// TwinCAT 3 PLC project plc_kfe_gatt
// Title: KFE GATT
// Company: LCLS - ECS
// ProjectVersion: 0.3.1
// ProgramVersion: 3.1.4023.0
// CompilerDefines: K
// libraries:
//   LCLS General, * (SLAC)
//   LCLS Vacuum, * (SLAC - LCLS)
//   lcls-twincat-motion, * (SLAC)
//   PMPS, * (SLAC - LCLS)
//   Tc2_ControllerToolbox, * (Beckhoff Automation GmbH)
//   Tc2_EtherCAT, * (Beckhoff Automation GmbH)
//   Tc2_MC2, * (Beckhoff Automation GmbH)
//   Tc2_Standard, * (Beckhoff Automation GmbH)
//   Tc2_System, * (Beckhoff Automation GmbH)
//   Tc2_Utilities, * (Beckhoff Automation GmbH)
//   Tc3_JsonXml, * (Beckhoff Automation GmbH)
//   Tc3_Module, * (Beckhoff Automation GmbH)
//   TcUnit, * (www.tcunit.org)
// project tree:
//   DUTs/ E_State.TcDUT, E_GasType.TcDUT, E_HomeState.TcDUT, E_MAA_States.TcDUT, E_MAA_States_X.TcDUT, E_MoveState.TcDUT, ST_DRL.TcDUT, ST_VGP.TcDUT
//   Version/ Global_Version.TcGVL
//   GVLs/ GVL_Devices.TcGVL, GVL_GATT.TcGVL, GVL_PMPS.TcGVL, GVL_MOT.TcGVL, GVL_Variables.TcGVL, Main.TcGVL
//   / PlcTask.TcTTO
//   POUs/ DIAGNOSTICS.TcPOU, FB_MAA.TcPOU, FB_MAA_States.TcPOU, FB_MAA_States_X.TcPOU, FB_VGP.TcPOU, PRG_1_PlcTask.TcPOU, PRG_GasSelection.TcPOU, PRG_GATT.TcPOU, PRG_ILK.TcPOU, PRG_INJ.TcPOU, PRG_Motion.TcPOU, PRG_Motors_Test.TcPOU, PRG_PMPS.TcPOU, PRG_Transmission.TcPOU, PRG_VGP.TcPOU
//   POUs/Test/ FB_ILK_TEST.TcPOU, FB_VCN_Lin.TcPOU
//   POUs/Transmission/ F_COEF_AR.TcPOU
// real-time tasks:
//   TASK PlcTask: cycle T#10ms, priority 20, ADS port 350
// motion (NC):
//   TASK NC-Task 1 SAF: cycle T#2ms, priority 4, ADS port 501
//   TASK NC-Task 1 SVB: cycle T#10ms, priority 8, ADS port 511
//   AXIS MA_1_X (id 1)
//     Velo: Maximum=1
//     OtherSettings: AllowMotionCmdToSlave=true
//     encoder EncType=7
//       EncPara: ScaleFactorNumerator=0.000117010498, Offset=1.88, Inverse=true, MaxCount=#x0000ffff, ReferenceSystem=1
//         SoftEndMinControl: Enable=true, Range=-2
//         SoftEndMaxControl: Enable=true, Range=2
//         Inc: RefSoftSyncMask=#x0000ffff
//     drive DrvType=24
//       Analog: VeloReferenz=7.93496, TorqueScale=10, ScaleFactorActTorque=0.1
//       TimeComp: TaskDelayCycles=1
//     controller CtrType=1
//       CtrPara: PriorControlFactor=1
//         PosDiffControl: Range=0.2
//         Observer: BandWidth=20
//   AXIS MA_1_Y (id 2)
//     Dynamic: AccelerationMaximum=30, DecelerationMaximum=30
//     Velo: Maximum=10
//     TargetPosControl: Range=0.5
//     OtherSettings: AllowMotionCmdToSlave=true
//     encoder EncType=7
//       EncPara: ScaleFactorNumerator=0.001490478515625, Offset=-48.83, MaxCount=#x0000ffff, ReferenceSystem=1
//         SoftEndMinControl: Enable=true, Range=-48.8
//         SoftEndMaxControl: Enable=true
//         Inc: RefSoftSyncMask=#x0000ffff
//     drive DrvType=24
//       Analog: VeloReferenz=40, TorqueScale=10, ScaleFactorActTorque=0.1
//       TimeComp: TaskDelayCycles=1
//     controller CtrType=1
//       CtrPara: PriorControlFactor=1
//         PosDiffControl: Range=0.5
//         Observer: BandWidth=20
//   AXIS MA_2_X (id 3)
//     Velo: Maximum=1
//     OtherSettings: AllowMotionCmdToSlave=true
//     encoder EncType=7
//       EncPara: ScaleFactorNumerator=7.6080322266e-05, Offset=-0.496, MaxCount=#x0000ffff, ReferenceSystem=1
//         SoftEndMinControl: Enable=true, Range=-1.59
//         SoftEndMaxControl: Enable=true, Range=1.59
//         Inc: RefSoftSyncMask=#x0000ffff
//     drive DrvType=24
//       Analog: VeloReferenz=7.93496, TorqueScale=10, ScaleFactorActTorque=0.1
//       TimeComp: TaskDelayCycles=1
//     controller CtrType=1
//       CtrPara: PriorControlFactor=1
//         PosDiffControl: Range=0.1
//         Observer: BandWidth=20
//   AXIS MA_2_Y (id 4)
//     Dynamic: AccelerationMaximum=30, DecelerationMaximum=30
//     Velo: Maximum=10
//     TargetPosControl: Range=0.5
//     OtherSettings: AllowMotionCmdToSlave=true
//     encoder EncType=7
//       EncPara: ScaleFactorNumerator=0.001524353027344, Offset=-49.38, MaxCount=#x0000ffff, ReferenceSystem=1
//         SoftEndMinControl: Enable=true, Range=-48.99
//         SoftEndMaxControl: Enable=true
//         Inc: RefSoftSyncMask=#x0000ffff
//     drive DrvType=24
//       Analog: VeloReferenz=50, TorqueScale=10, ScaleFactorActTorque=0.1
//       TimeComp: TaskDelayCycles=1
//     controller CtrType=1
//       CtrPara: PriorControlFactor=1
//         PosDiffControl: Range=0.5
//         Observer: BandWidth=20
//   AXIS MA_3_X (id 5)
//     Velo: Maximum=1
//     OtherSettings: AllowMotionCmdToSlave=true
//     encoder EncType=7
//       EncPara: ScaleFactorNumerator=0.0001220703125, Offset=-2.029, MaxCount=#x0000ffff, ReferenceSystem=1
//         SoftEndMinControl: Enable=true, Range=-1.6
//         SoftEndMaxControl: Enable=true, Range=1.6
//         Inc: RefSoftSyncMask=#x0000ffff
//     drive DrvType=24
//       Analog: VeloReferenz=7.93496, TorqueScale=10, ScaleFactorActTorque=0.1
//       TimeComp: TaskDelayCycles=1
//     controller CtrType=1
//       CtrPara: PriorControlFactor=1
//         PosDiffControl: Range=0.1
//         Observer: BandWidth=20
//   AXIS MA_3_Y (id 6)
//     Dynamic: AccelerationMaximum=30, DecelerationMaximum=30
//     Velo: Maximum=10
//     TargetPosControl: Range=0.5
//     OtherSettings: AllowMotionCmdToSlave=true
//     encoder EncType=7
//       EncPara: ScaleFactorNumerator=0.001514892578125, Offset=-49.49, MaxCount=#x0000ffff, ReferenceSystem=1
//         SoftEndMinControl: Enable=true, Range=-49.27
//         SoftEndMaxControl: Enable=true
//         Inc: RefSoftSyncMask=#x0000ffff
//     drive DrvType=24
//       Analog: VeloReferenz=50, TorqueScale=10, ScaleFactorActTorque=0.1
//       TimeComp: TaskDelayCycles=1
//     controller CtrType=1
//       CtrPara: PriorControlFactor=1
//         PosDiffControl: Range=0.2
//         Observer: BandWidth=20
//   AXIS MA_4_X (id 7)
//     Velo: Maximum=1
//     OtherSettings: AllowMotionCmdToSlave=true
//     encoder EncType=7
//       EncPara: ScaleFactorNumerator=0.0001022338867, Offset=-1.581, MaxCount=#x0000ffff, ReferenceSystem=1
//         SoftEndMinControl: Enable=true, Range=-1.58
//         SoftEndMaxControl: Enable=true, Range=1.76
//         Inc: RefSoftSyncMask=#x0000ffff
//     drive DrvType=24
//       Analog: VeloReferenz=7.93496, TorqueScale=10, ScaleFactorActTorque=0.1
//       TimeComp: TaskDelayCycles=1
//     controller CtrType=1
//       CtrPara: PriorControlFactor=1
//         PosDiffControl: Range=0.2
//         Observer: BandWidth=20
//   AXIS MA_4_Y (id 8)
//     Dynamic: AccelerationMaximum=30, DecelerationMaximum=30
//     Velo: Maximum=10
//     TargetPosControl: Range=0.5
//     OtherSettings: AllowMotionCmdToSlave=true
//     encoder EncType=7
//       EncPara: ScaleFactorNumerator=0.001497802734375, Offset=-49.07, MaxCount=#x0000ffff, ReferenceSystem=1
//         SoftEndMinControl: Enable=true, Range=-49.08
//         SoftEndMaxControl: Enable=true, Range=0.009
//         Inc: RefSoftSyncMask=#x0000ffff
//     drive DrvType=24
//       Analog: VeloReferenz=50, TorqueScale=10, ScaleFactorActTorque=0.1
//       TimeComp: TaskDelayCycles=1
//     controller CtrType=1
//       CtrPara: PriorControlFactor=1
//         PosDiffControl: Range=0.2
//         Observer: BandWidth=20
//   AXIS VGP_80 (id 9)
//     Velo: Maximum=1800
//     OtherSettings: AllowMotionCmdToSlave=true
//     encoder EncType=4
//       EncPara: ScaleFactorNumerator=0.0390625, Inverse=true, MaxCount=#x0000ffff
//         SoftEndMinControl: Enable=true, Range=-15
//         SoftEndMaxControl: Enable=true, Range=1680
//         Inc: RefSoftSyncMask=#x0000ffff
//     drive DrvType=24
//       Analog: VeloReferenz=1000, TorqueScale=10, ScaleFactorActTorque=0.1
//       TimeComp: TaskDelayCycles=1
//     controller CtrType=1
//       CtrPara: PriorControlFactor=1
//         PosDiffControl: Range=10
//         Observer: BandWidth=20
// I/O:
//   DEVICE =+-CX2020/EtherCAT1, AmsNetId 172.21.92.57.2.1
//     =+-EK1200_00_00 [EK1200-5000 EtherCAT Power supply (2A E-Bus)]
//       =+-ES3064_00_01 [EL3064 4Ch. Ana. Input 0-10V]
//       =+-EL6070_00_02 [EL6070 1Ch. Licensing-Terminal]
//       =+-ES1008_00_03 [EL1008 8Ch. Dig. Input 24V, 3ms]
//       =+-ES2008_00_05 [EL2008 8Ch. Dig. Output 24V, 0.5A]
//       =+-EL2794_00_06 [EL2794 4Ch. Dig. Output 24V AC/DC, 2A, short-circuit-proof]
//       =+-ES2202_00_07 [EL2202 2Ch. Dig. Output 24V, 0.5A]
//       PMPS_PRE [EL6695 EtherCAT Bridge terminal (Primary)]
//       =+-EK1110_00_09 [EK1110 EtherCAT extension]
//     =+-EK1100_01_00 [EK1100 EtherCAT Coupler (2A E-Bus)]
//       =+-ES3064_01_01 [EL3064 4Ch. Ana. Input 0-10V]
//       =+-ES3064_01_02 [EL3064 4Ch. Ana. Input 0-10V]
//       =+-EL2798_01_03 [EL2798 8Ch. Dig. Output 24V AC/DC, 2A, potential-free]
//       =+-ES3064_01_04 [EL3064 4Ch. Ana. Input 0-10V]
//       =+-ES3064_01_05 [EL3064 4Ch. Ana. Input 0-10V]
//       =+-ES3064_01_06 [EL3064 4Ch. Ana. Input 0-10V]
//       =+-ES3064_01_07 [EL3064 4Ch. Ana. Input 0-10V]
//       =+-EL2798_01_08 [EL2798 8Ch. Dig. Output 24V AC/DC, 2A, potential-free]
//       =+-ES3064_01_09 [EL3064 4Ch. Ana. Input 0-10V]
//       =+-ES3064_01_10 [EL3064 4Ch. Ana. Input 0-10V]
//       =+-EL9410_01_11 [EL9410 E-Bus Power Supplier  (Diagnostics)]
//       =+-ES3064_01_12 [EL3064 4Ch. Ana. Input 0-10V]
//       =+-ES3064_01_13 [EL3064 4Ch. Ana. Input 0-10V]
//       =+-EL2798_01_14 [EL2798 8Ch. Dig. Output 24V AC/DC, 2A, potential-free]
//       =+-ES3064_01_15 [EL3064 4Ch. Ana. Input 0-10V]
//       =+-ES3064_01_16 [EL3064 4Ch. Ana. Input 0-10V]
//       =+-ES3064_01_17 [EL3064 4Ch. Ana. Input 0-10V]
//       =+-ES3064_01_18 [EL3064 4Ch. Ana. Input 0-10V]
//       =+-EL2798_01_19 [EL2798 8Ch. Dig. Output 24V AC/DC, 2A, potential-free]
//       =+-ES3064_01_20 [EL3064 4Ch. Ana. Input 0-10V]
//       =+-ES3064_01_21 [EL3064 4Ch. Ana. Input 0-10V]
//       =+-EK1110_01_22 [EK1110 EtherCAT extension]
//     =+-EK1100_02_00 [EK1100 EtherCAT Coupler (2A E-Bus)]
//       =+-ES2004_02_01 [EL2004 4Ch. Dig. Output 24V, 0.5A]
//       =+-ES1004_02_02 [EL1004 4Ch. Dig. Input 24V, 3ms]
//       =+-ES2004_02_03 [EL2004 4Ch. Dig. Output 24V, 0.5A]
//       =+-ES1004_02_04 [EL1004 4Ch. Dig. Input 24V, 3ms]
//       =+-ES7041_02_05 [EL7041 1Ch. Stepper motor output stage (50V, 5A)]
//       =+-ES7041_02_06 [EL7041 1Ch. Stepper motor output stage (50V, 5A)]
//       =+-ES2004_02_07 [EL2004 4Ch. Dig. Output 24V, 0.5A]
//       =+-ES1004_02_08 [EL1004 4Ch. Dig. Input 24V, 3ms]
//       =+-ES7041_02_09 [EL7041 1Ch. Stepper motor output stage (50V, 5A)]
//       =+-ES7041_02_10 [EL7041 1Ch. Stepper motor output stage (50V, 5A)]
//       =+-ES3064_02_11 [EL3064 4Ch. Ana. Input 0-10V]
//       =+-ES9070_02_12 [EL9070 Shield terminal]
//       =+-ES1008_02_13 [EL1008 8Ch. Dig. Input 24V, 3ms]
//       =+-ES2008_02_14 [EL2008 8Ch. Dig. Output 24V, 0.5A]
//       =+-EL2794_02_15 [EL2794 4Ch. Dig. Output 24V AC/DC, 2A, short-circuit-proof]
//       =+-EL9184_02_16 [EL9184 Potential Connection, 8 x 24V, 8 x Ground]
//       =+-ES3054_02_17 [EL3054 4Ch. Ana. Input 4-20mA]
//       =+-ES6021_02_18 [EL6021 Interface (RS422/485)]
//       =+-EL9011_02_19 [EL9011 End Terminal]
//     =+-EK1100_03_00 [EK1100 EtherCAT Coupler (2A E-Bus)]
//       =+-ES1004_03_01 [EL1004 4Ch. Dig. Input 24V, 3ms]
//       =+-ES1004_03_02 [EL1004 4Ch. Dig. Input 24V, 3ms]
//       =+-EL2798_03_03 [EL2798 8Ch. Dig. Output 24V AC/DC, 2A, potential-free]
//       =+-ES3064_03_04 [EL3064 4Ch. Ana. Input 0-10V]
//       =+-ES4004_03_05 [EL4004 4Ch. Ana. Output 0-10V, 12bit]
//       =+-ES3064_03_06 [EL3064 4Ch. Ana. Input 0-10V]
//       =+-EL2798_03_07 [EL2798 8Ch. Dig. Output 24V AC/DC, 2A, potential-free]
//       =+-ES1004_03_08 [EL1004 4Ch. Dig. Input 24V, 3ms]
//       =+-ES1004_03_09 [EL1004 4Ch. Dig. Input 24V, 3ms]
//       =+-EL9410_03_10 [EL9410 E-Bus Power Supplier  (Diagnostics)]
//       =+-ES1004_03_11 [EL1004 4Ch. Dig. Input 24V, 3ms]
//       =+-ES1004_03_12 [EL1004 4Ch. Dig. Input 24V, 3ms]
//       =+-EL2798_03_13 [EL2798 8Ch. Dig. Output 24V AC/DC, 2A, potential-free]
//       =+-ES3064_03_14 [EL3064 4Ch. Ana. Input 0-10V]
//       =+-ES4004_03_15 [EL4004 4Ch. Ana. Output 0-10V, 12bit]
//       =+-ES3064_03_16 [EL3064 4Ch. Ana. Input 0-10V]
//       =+-EL2798_03_17 [EL2798 8Ch. Dig. Output 24V AC/DC, 2A, potential-free]
//       =+-ES1004_03_18 [EL1004 4Ch. Dig. Input 24V, 3ms]
//       =+-ES1004_03_19 [EL1004 4Ch. Dig. Input 24V, 3ms]
//       =+-EL2794_03_20 [EL2794 4Ch. Dig. Output 24V AC/DC, 2A, short-circuit-proof]
//       =+-ES1004_03_21 [EL1004 4Ch. Dig. Input 24V, 3ms]
//       =+-EL9011_03_22 [EL9011 End Terminal]
//     =+-EK1100_04_00 [EK1100 EtherCAT Coupler (2A E-Bus)]
//       =+-ES2004_04_01 [EL2004 4Ch. Dig. Output 24V, 0.5A]
//       =+-ES4004_04_02 [EL4004 4Ch. Ana. Output 0-10V, 12bit]
//       =+-EL9184_04_03 [EL9184 Potential Connection, 8 x 24V, 8 x Ground]
//       =+-EL7041_04_04
//       =+-EL5101_04_05
//       =+-ES1084_04_06 [EL1084 4Ch. Dig. Input 24V, 3ms, negative]
//       =+-EL7041_04_07 [EL7041 1Ch. Stepper motor output stage (50V, 5A)]
//       =+-EL7041_04_08 [EL7041 1Ch. Stepper motor output stage (50V, 5A)]
//       =+-ES2004_04_09 [EL2004 4Ch. Dig. Output 24V, 0.5A]
//       =+-EL7041_04_10 [EL7041 1Ch. Stepper motor output stage (50V, 5A)]
//       =+-EL7041_04_11 [EL7041 1Ch. Stepper motor output stage (50V, 5A)]
//       =+-ES3054_04_12 [EL3054 4Ch. Ana. Input 4-20mA]
//       =+-ES1084_04_13 [EL1084 4Ch. Dig. Input 24V, 3ms, negative]
//       =+-ES6021_04_14 [EL6021 Interface (RS422/485)]
//       =+-EL9184_04_15 [EL9184 Potential Connection, 8 x 24V, 8 x Ground]
//       =+-ES9070_04_16 [EL9070 Shield terminal]
//       =+-EL3174_04_17 [EL3174-0002 4Ch. Ana. Input +/-10V, +/-20mA 16 Bit, Isolated Channels]
//       =+-EL2212_04_18 [EL2212 2Ch. dig. output with overexcitation (24V DC, 2.5A, 10A Peak)]
//       =+-EL9011_04_19 [EL9011 End Terminal]
//     =+-EK1100_05_00 [EK1100 EtherCAT Coupler (2A E-Bus)]
//       =+-ES1004_05_01 [EL1004 4Ch. Dig. Input 24V, 3ms]
//       =+-ES2004_05_02 [EL2004 4Ch. Dig. Output 24V, 0.5A]
//       =+-ES1004_05_03 [EL1004 4Ch. Dig. Input 24V, 3ms]
//       =+-ES2004_05_04 [EL2004 4Ch. Dig. Output 24V, 0.5A]
//       =+-ES2004_05_05 [EL2004 4Ch. Dig. Output 24V, 0.5A]
//       =+-ES1004_05_06 [EL1004 4Ch. Dig. Input 24V, 3ms]
//       =+-ES2004_05_07 [EL2004 4Ch. Dig. Output 24V, 0.5A]
//       =+-ES1004_05_08 [EL1004 4Ch. Dig. Input 24V, 3ms]
//       =+-EL2212_05_09 [EL2212 2Ch. dig. output with overexcitation (24V DC, 2.5A, 10A Peak)]
//       =+-EL2798_05_10 [EL2798 8Ch. Dig. Output 24V AC/DC, 2A, potential-free]
//       =+-ES1004_05_11 [EL1004 4Ch. Dig. Input 24V, 3ms]
//       =+-EL1084_05_12 [EL1084 4Ch. Dig. Input 24V, 3ms, negative]
//       =+-EL1084_05_13 [EL1084 4Ch. Dig. Input 24V, 3ms, negative]
//       =+-EL9184_05_14 [EL9184 Potential Connection, 8 x 24V, 8 x Ground]
//       =+-ES9070_05_15 [EL9070 Shield terminal]
//       =+-EL3174_05_16 [EL3174-0002 4Ch. Ana. Input +/-10V, +/-20mA 16 Bit, Isolated Channels]
//       =+-EL9011_05_17 [EL9011 End Terminal]
//     =+-EK1100_06_00 [EK1100 EtherCAT Coupler (2A E-Bus)]
//       =+-ES1004_06_01 [EL1004 4Ch. Dig. Input 24V, 3ms]
//       =+-ES1004_06_02 [EL1004 4Ch. Dig. Input 24V, 3ms]
//       =+-EL2798_06_03 [EL2798 8Ch. Dig. Output 24V AC/DC, 2A, potential-free]
//       =+-ES3064_06_04 [EL3064 4Ch. Ana. Input 0-10V]
//       =+-ES4004_06_05 [EL4004 4Ch. Ana. Output 0-10V, 12bit]
//       =+-ES3064_06_06 [EL3064 4Ch. Ana. Input 0-10V]
//       =+-EL2798_06_07 [EL2798 8Ch. Dig. Output 24V AC/DC, 2A, potential-free]
//       =+-ES1004_06_08 [EL1004 4Ch. Dig. Input 24V, 3ms]
//       =+-ES1004_06_09 [EL1004 4Ch. Dig. Input 24V, 3ms]
//       =+-EL9410_06_10 [EL9410 E-Bus Power Supplier  (Diagnostics)]
//       =+-ES1004_06_11 [EL1004 4Ch. Dig. Input 24V, 3ms]
//       =+-ES1004_06_12 [EL1004 4Ch. Dig. Input 24V, 3ms]
//       =+-EL2798_06_13 [EL2798 8Ch. Dig. Output 24V AC/DC, 2A, potential-free]
//       =+-ES3064_06_14 [EL3064 4Ch. Ana. Input 0-10V]
//       =+-ES4004_06_15 [EL4004 4Ch. Ana. Output 0-10V, 12bit]
//       =+-ES3064_06_16 [EL3064 4Ch. Ana. Input 0-10V]
//       =+-EL2798_06_17 [EL2798 8Ch. Dig. Output 24V AC/DC, 2A, potential-free]
//       =+-ES1004_06_18 [EL1004 4Ch. Dig. Input 24V, 3ms]
//       =+-ES1004_06_19 [EL1004 4Ch. Dig. Input 24V, 3ms]
//       =+-ES1088_06_20 [EL1088 8Ch. Dig. Input 24V, 3ms, negative]
//       =+-ES9187_06_21 [EL9187 Potential Connection, 8 x Ground]
//       =+-EL2794_06_22 [EL2794 4Ch. Dig. Output 24V AC/DC, 2A, short-circuit-proof]
//       =+-ES1088_06_23 [EL1088 8Ch. Dig. Input 24V, 3ms, negative]
//       =+-ES9187_06_24 [EL9187 Potential Connection, 8 x Ground]
//       =+-EL2212_06_25 [EL2212 2Ch. dig. output with overexcitation (24V DC, 2.5A, 10A Peak)]
//       =+-EL9011_06_26 [EL9011 End Terminal]
// variable links:
//   NC-Task 1 SAF/Axes/MA_1_X <-> =+-CX2020/EtherCAT1/=+-EK1100_02_00/=+-ES3054_02_17
//     Enc/Inputs/In/nDataIn1[0] <-> AI Standard Channel 1/Value
//     Enc/Inputs/In/nState4 @bit 1 <-> WcState/InputToggle
//     Enc/Inputs/In/nState4 <-> WcState/WcState
//   NC-Task 1 SAF/Axes/MA_1_X <-> =+-CX2020/EtherCAT1/=+-EK1100_02_00/=+-ES7041_02_05
//     Drive/Inputs/In/nState1 @bit 3 <-> STM Status/Status/Error
//     Drive/Inputs/In/nState1 @bit 5 <-> STM Status/Status/Moving negative
//     Drive/Inputs/In/nState1 @bit 4 <-> STM Status/Status/Moving positive
//     Drive/Inputs/In/nState1 @bit 1 <-> STM Status/Status/Ready
//     Drive/Inputs/In/nState1 <-> STM Status/Status/Ready to enable
//     Drive/Inputs/In/nState1 @bit 6 <-> STM Status/Status/Torque reduced
//     Drive/Inputs/In/nState1 @bit 2 <-> STM Status/Status/Warning
//     Drive/Inputs/In/nState2 @bit 3 <-> STM Status/Status/Digital input 1
//     Drive/Inputs/In/nState2 @bit 4 <-> STM Status/Status/Digital input 2
//     Drive/Inputs/In/nState2 @bit 5 <-> STM Status/Status/Sync error
//     Drive/Inputs/In/nState2 @bit 7 <-> STM Status/Status/TxPDO Toggle
//     Drive/Inputs/In/nState4 @bit 1 <-> WcState/InputToggle
//     Drive/Inputs/In/nState4 <-> WcState/WcState
//     Drive/Outputs/Out/nCtrl1 <-> STM Control/Control/Enable
//     Drive/Outputs/Out/nCtrl1 @bit 2 <-> STM Control/Control/Reduce torque
//     Drive/Outputs/Out/nCtrl1 @bit 1 <-> STM Control/Control/Reset
//     Drive/Outputs/Out/nDataOut2[0] <-> STM Velocity/Velocity
//   NC-Task 1 SAF/Axes/MA_1_Y <-> =+-CX2020/EtherCAT1/=+-EK1100_02_00/=+-ES3054_02_17
//     Enc/Inputs/In/nDataIn1[0] <-> AI Standard Channel 2/Value
//     Enc/Inputs/In/nState4 @bit 1 <-> WcState/InputToggle
//     Enc/Inputs/In/nState4 <-> WcState/WcState
//   NC-Task 1 SAF/Axes/MA_1_Y <-> =+-CX2020/EtherCAT1/=+-EK1100_02_00/=+-ES7041_02_06
//     Drive/Inputs/In/nState1 @bit 3 <-> STM Status/Status/Error
//     Drive/Inputs/In/nState1 @bit 5 <-> STM Status/Status/Moving negative
//     Drive/Inputs/In/nState1 @bit 4 <-> STM Status/Status/Moving positive
//     Drive/Inputs/In/nState1 @bit 1 <-> STM Status/Status/Ready
//     Drive/Inputs/In/nState1 <-> STM Status/Status/Ready to enable
//     Drive/Inputs/In/nState1 @bit 6 <-> STM Status/Status/Torque reduced
//     Drive/Inputs/In/nState1 @bit 2 <-> STM Status/Status/Warning
//     Drive/Inputs/In/nState2 @bit 3 <-> STM Status/Status/Digital input 1
//     Drive/Inputs/In/nState2 @bit 4 <-> STM Status/Status/Digital input 2
//     Drive/Inputs/In/nState2 @bit 5 <-> STM Status/Status/Sync error
//     Drive/Inputs/In/nState2 @bit 7 <-> STM Status/Status/TxPDO Toggle
//     Drive/Inputs/In/nState4 @bit 1 <-> WcState/InputToggle
//     Drive/Inputs/In/nState4 <-> WcState/WcState
//     Drive/Outputs/Out/nCtrl1 <-> STM Control/Control/Enable
//     Drive/Outputs/Out/nCtrl1 @bit 2 <-> STM Control/Control/Reduce torque
//     Drive/Outputs/Out/nCtrl1 @bit 1 <-> STM Control/Control/Reset
//     Drive/Outputs/Out/nDataOut2[0] <-> STM Velocity/Velocity
//   NC-Task 1 SAF/Axes/MA_2_X <-> =+-CX2020/EtherCAT1/=+-EK1100_02_00/=+-ES3054_02_17
//     Enc/Inputs/In/nDataIn1[0] <-> AI Standard Channel 3/Value
//     Enc/Inputs/In/nState4 @bit 1 <-> WcState/InputToggle
//     Enc/Inputs/In/nState4 <-> WcState/WcState
//   NC-Task 1 SAF/Axes/MA_2_X <-> =+-CX2020/EtherCAT1/=+-EK1100_02_00/=+-ES7041_02_09
//     Drive/Inputs/In/nState1 @bit 3 <-> STM Status/Status/Error
//     Drive/Inputs/In/nState1 @bit 5 <-> STM Status/Status/Moving negative
//     Drive/Inputs/In/nState1 @bit 4 <-> STM Status/Status/Moving positive
//     Drive/Inputs/In/nState1 @bit 1 <-> STM Status/Status/Ready
//     Drive/Inputs/In/nState1 <-> STM Status/Status/Ready to enable
//     Drive/Inputs/In/nState1 @bit 6 <-> STM Status/Status/Torque reduced
//     Drive/Inputs/In/nState1 @bit 2 <-> STM Status/Status/Warning
//     Drive/Inputs/In/nState2 @bit 3 <-> STM Status/Status/Digital input 1
//     Drive/Inputs/In/nState2 @bit 4 <-> STM Status/Status/Digital input 2
//     Drive/Inputs/In/nState2 @bit 5 <-> STM Status/Status/Sync error
//     Drive/Inputs/In/nState2 @bit 7 <-> STM Status/Status/TxPDO Toggle
//     Drive/Inputs/In/nState4 @bit 1 <-> WcState/InputToggle
//     Drive/Inputs/In/nState4 <-> WcState/WcState
//     Drive/Outputs/Out/nCtrl1 <-> STM Control/Control/Enable
//     Drive/Outputs/Out/nCtrl1 @bit 2 <-> STM Control/Control/Reduce torque
//     Drive/Outputs/Out/nCtrl1 @bit 1 <-> STM Control/Control/Reset
//     Drive/Outputs/Out/nDataOut2[0] <-> STM Velocity/Velocity
//   NC-Task 1 SAF/Axes/MA_2_Y <-> =+-CX2020/EtherCAT1/=+-EK1100_02_00/=+-ES3054_02_17
//     Enc/Inputs/In/nDataIn1[0] <-> AI Standard Channel 4/Value
//     Enc/Inputs/In/nState4 @bit 1 <-> WcState/InputToggle
//     Enc/Inputs/In/nState4 <-> WcState/WcState
//   NC-Task 1 SAF/Axes/MA_2_Y <-> =+-CX2020/EtherCAT1/=+-EK1100_02_00/=+-ES7041_02_10
//     Drive/Inputs/In/nState1 @bit 3 <-> STM Status/Status/Error
//     Drive/Inputs/In/nState1 @bit 5 <-> STM Status/Status/Moving negative
//     Drive/Inputs/In/nState1 @bit 4 <-> STM Status/Status/Moving positive
//     Drive/Inputs/In/nState1 @bit 1 <-> STM Status/Status/Ready
//     Drive/Inputs/In/nState1 <-> STM Status/Status/Ready to enable
//     Drive/Inputs/In/nState1 @bit 6 <-> STM Status/Status/Torque reduced
//     Drive/Inputs/In/nState1 @bit 2 <-> STM Status/Status/Warning
//     Drive/Inputs/In/nState2 @bit 3 <-> STM Status/Status/Digital input 1
//     Drive/Inputs/In/nState2 @bit 4 <-> STM Status/Status/Digital input 2
//     Drive/Inputs/In/nState2 @bit 5 <-> STM Status/Status/Sync error
//     Drive/Inputs/In/nState2 @bit 7 <-> STM Status/Status/TxPDO Toggle
//     Drive/Inputs/In/nState4 @bit 1 <-> WcState/InputToggle
//     Drive/Inputs/In/nState4 <-> WcState/WcState
//     Drive/Outputs/Out/nCtrl1 <-> STM Control/Control/Enable
//     Drive/Outputs/Out/nCtrl1 @bit 2 <-> STM Control/Control/Reduce torque
//     Drive/Outputs/Out/nCtrl1 @bit 1 <-> STM Control/Control/Reset
//     Drive/Outputs/Out/nDataOut2[0] <-> STM Velocity/Velocity
//   NC-Task 1 SAF/Axes/MA_3_X <-> =+-CX2020/EtherCAT1/=+-EK1100_04_00/=+-EL7041_04_07
//     Drive/Inputs/In/nState1 @bit 3 <-> STM Status/Status/Error
//     Drive/Inputs/In/nState1 @bit 5 <-> STM Status/Status/Moving negative
//     Drive/Inputs/In/nState1 @bit 4 <-> STM Status/Status/Moving positive
//     Drive/Inputs/In/nState1 @bit 1 <-> STM Status/Status/Ready
//     Drive/Inputs/In/nState1 <-> STM Status/Status/Ready to enable
//     Drive/Inputs/In/nState1 @bit 6 <-> STM Status/Status/Torque reduced
//     Drive/Inputs/In/nState1 @bit 2 <-> STM Status/Status/Warning
//     Drive/Inputs/In/nState2 @bit 3 <-> STM Status/Status/Digital input 1
//     Drive/Inputs/In/nState2 @bit 4 <-> STM Status/Status/Digital input 2
//     Drive/Inputs/In/nState2 @bit 5 <-> STM Status/Status/Sync error
//     Drive/Inputs/In/nState2 @bit 7 <-> STM Status/Status/TxPDO Toggle
//     Drive/Inputs/In/nState4 @bit 1 <-> WcState/InputToggle
//     Drive/Inputs/In/nState4 <-> WcState/WcState
//     Drive/Outputs/Out/nCtrl1 <-> STM Control/Control/Enable
//     Drive/Outputs/Out/nCtrl1 @bit 2 <-> STM Control/Control/Reduce torque
//     Drive/Outputs/Out/nCtrl1 @bit 1 <-> STM Control/Control/Reset
//     Drive/Outputs/Out/nDataOut2[0] <-> STM Velocity/Velocity
//   NC-Task 1 SAF/Axes/MA_3_X <-> =+-CX2020/EtherCAT1/=+-EK1100_04_00/=+-ES3054_04_12
//     Enc/Inputs/In/nDataIn1[0] <-> AI Standard Channel 1/Value
//     Enc/Inputs/In/nState4 @bit 1 <-> WcState/InputToggle
//     Enc/Inputs/In/nState4 <-> WcState/WcState
//   NC-Task 1 SAF/Axes/MA_3_Y <-> =+-CX2020/EtherCAT1/=+-EK1100_04_00/=+-EL7041_04_08
//     Drive/Inputs/In/nState1 @bit 3 <-> STM Status/Status/Error
//     Drive/Inputs/In/nState1 @bit 5 <-> STM Status/Status/Moving negative
//     Drive/Inputs/In/nState1 @bit 4 <-> STM Status/Status/Moving positive
//     Drive/Inputs/In/nState1 @bit 1 <-> STM Status/Status/Ready
//     Drive/Inputs/In/nState1 <-> STM Status/Status/Ready to enable
//     Drive/Inputs/In/nState1 @bit 6 <-> STM Status/Status/Torque reduced
//     Drive/Inputs/In/nState1 @bit 2 <-> STM Status/Status/Warning
//     Drive/Inputs/In/nState2 @bit 3 <-> STM Status/Status/Digital input 1
//     Drive/Inputs/In/nState2 @bit 4 <-> STM Status/Status/Digital input 2
//     Drive/Inputs/In/nState2 @bit 5 <-> STM Status/Status/Sync error
//     Drive/Inputs/In/nState2 @bit 7 <-> STM Status/Status/TxPDO Toggle
//     Drive/Inputs/In/nState4 @bit 1 <-> WcState/InputToggle
//     Drive/Inputs/In/nState4 <-> WcState/WcState
//     Drive/Outputs/Out/nCtrl1 <-> STM Control/Control/Enable
//     Drive/Outputs/Out/nCtrl1 @bit 2 <-> STM Control/Control/Reduce torque
//     Drive/Outputs/Out/nCtrl1 @bit 1 <-> STM Control/Control/Reset
//     Drive/Outputs/Out/nDataOut2[0] <-> STM Velocity/Velocity
//   NC-Task 1 SAF/Axes/MA_3_Y <-> =+-CX2020/EtherCAT1/=+-EK1100_04_00/=+-ES3054_04_12
//     Enc/Inputs/In/nDataIn1[0] <-> AI Standard Channel 2/Value
//     Enc/Inputs/In/nState4 @bit 1 <-> WcState/InputToggle
//     Enc/Inputs/In/nState4 <-> WcState/WcState
//   NC-Task 1 SAF/Axes/MA_4_X <-> =+-CX2020/EtherCAT1/=+-EK1100_04_00/=+-EL7041_04_10
//     Drive/Inputs/In/nState1 @bit 3 <-> STM Status/Status/Error
//     Drive/Inputs/In/nState1 @bit 5 <-> STM Status/Status/Moving negative
//     Drive/Inputs/In/nState1 @bit 4 <-> STM Status/Status/Moving positive
//     Drive/Inputs/In/nState1 @bit 1 <-> STM Status/Status/Ready
//     Drive/Inputs/In/nState1 <-> STM Status/Status/Ready to enable
//     Drive/Inputs/In/nState1 @bit 6 <-> STM Status/Status/Torque reduced
//     Drive/Inputs/In/nState1 @bit 2 <-> STM Status/Status/Warning
//     Drive/Inputs/In/nState2 @bit 3 <-> STM Status/Status/Digital input 1
//     Drive/Inputs/In/nState2 @bit 4 <-> STM Status/Status/Digital input 2
//     Drive/Inputs/In/nState2 @bit 5 <-> STM Status/Status/Sync error
//     Drive/Inputs/In/nState2 @bit 7 <-> STM Status/Status/TxPDO Toggle
//     Drive/Inputs/In/nState4 @bit 1 <-> WcState/InputToggle
//     Drive/Inputs/In/nState4 <-> WcState/WcState
//     Drive/Outputs/Out/nCtrl1 <-> STM Control/Control/Enable
//     Drive/Outputs/Out/nCtrl1 @bit 2 <-> STM Control/Control/Reduce torque
//     Drive/Outputs/Out/nCtrl1 @bit 1 <-> STM Control/Control/Reset
//     Drive/Outputs/Out/nDataOut2[0] <-> STM Velocity/Velocity
//   NC-Task 1 SAF/Axes/MA_4_X <-> =+-CX2020/EtherCAT1/=+-EK1100_04_00/=+-ES3054_04_12
//     Enc/Inputs/In/nDataIn1[0] <-> AI Standard Channel 3/Value
//     Enc/Inputs/In/nState4 @bit 1 <-> WcState/InputToggle
//     Enc/Inputs/In/nState4 <-> WcState/WcState
//   NC-Task 1 SAF/Axes/MA_4_Y <-> =+-CX2020/EtherCAT1/=+-EK1100_04_00/=+-EL7041_04_11
//     Drive/Inputs/In/nState1 @bit 3 <-> STM Status/Status/Error
//     Drive/Inputs/In/nState1 @bit 5 <-> STM Status/Status/Moving negative
//     Drive/Inputs/In/nState1 @bit 4 <-> STM Status/Status/Moving positive
//     Drive/Inputs/In/nState1 @bit 1 <-> STM Status/Status/Ready
//     Drive/Inputs/In/nState1 <-> STM Status/Status/Ready to enable
//     Drive/Inputs/In/nState1 @bit 6 <-> STM Status/Status/Torque reduced
//     Drive/Inputs/In/nState1 @bit 2 <-> STM Status/Status/Warning
//     Drive/Inputs/In/nState2 @bit 3 <-> STM Status/Status/Digital input 1
//     Drive/Inputs/In/nState2 @bit 4 <-> STM Status/Status/Digital input 2
//     Drive/Inputs/In/nState2 @bit 5 <-> STM Status/Status/Sync error
//     Drive/Inputs/In/nState2 @bit 7 <-> STM Status/Status/TxPDO Toggle
//     Drive/Inputs/In/nState4 @bit 1 <-> WcState/InputToggle
//     Drive/Inputs/In/nState4 <-> WcState/WcState
//     Drive/Outputs/Out/nCtrl1 <-> STM Control/Control/Enable
//     Drive/Outputs/Out/nCtrl1 @bit 2 <-> STM Control/Control/Reduce torque
//     Drive/Outputs/Out/nCtrl1 @bit 1 <-> STM Control/Control/Reset
//     Drive/Outputs/Out/nDataOut2[0] <-> STM Velocity/Velocity
//   NC-Task 1 SAF/Axes/MA_4_Y <-> =+-CX2020/EtherCAT1/=+-EK1100_04_00/=+-ES3054_04_12
//     Enc/Inputs/In/nDataIn1[0] <-> AI Standard Channel 4/Value
//     Enc/Inputs/In/nState4 @bit 1 <-> WcState/InputToggle
//     Enc/Inputs/In/nState4 <-> WcState/WcState
//   NC-Task 1 SAF/Axes/VGP_80 <-> =+-CX2020/EtherCAT1/=+-EK1100_04_00/=+-EL5101_04_05
//     Enc/Inputs/In/nDataIn1[0] <-> ENC Status compact/Counter value
//     Enc/Inputs/In/nDataIn2[0] <-> ENC Status compact/Latch value
//     Enc/Inputs/In/nState1 @bit 4 <-> ENC Status compact/Status/Counter overflow
//     Enc/Inputs/In/nState1 @bit 3 <-> ENC Status compact/Status/Counter underflow
//     Enc/Inputs/In/nState1 @bit 7 <-> ENC Status compact/Status/Extrapolation stall
//     Enc/Inputs/In/nState1 <-> ENC Status compact/Status/Latch C valid
//     Enc/Inputs/In/nState1 @bit 1 <-> ENC Status compact/Status/Latch extern valid
//     Enc/Inputs/In/nState1 @bit 6 <-> ENC Status compact/Status/Open circuit
//     Enc/Inputs/In/nState1 @bit 2 <-> ENC Status compact/Status/Set counter done
//     Enc/Inputs/In/nState1 @bit 5 <-> ENC Status compact/Status/Status of input status
//     Enc/Inputs/In/nState2 @bit 4 <-> ENC Status compact/Status/Status of extern latch
//     Enc/Inputs/In/nState2 <-> ENC Status compact/Status/Status of input A
//     Enc/Inputs/In/nState2 @bit 1 <-> ENC Status compact/Status/Status of input B
//     Enc/Inputs/In/nState2 @bit 2 <-> ENC Status compact/Status/Status of input C
//     Enc/Inputs/In/nState2 @bit 3 <-> ENC Status compact/Status/Status of input gate
//     Enc/Inputs/In/nState2 @bit 5 <-> ENC Status compact/Status/Sync error
//     Enc/Inputs/In/nState2 @bit 6 <-> ENC Status compact/Status/TxPDO State
//     Enc/Inputs/In/nState2 @bit 7 <-> ENC Status compact/Status/TxPDO Toggle
//     Enc/Inputs/In/nState4 @bit 1 <-> WcState/InputToggle
//     Enc/Inputs/In/nState4 <-> WcState/WcState
//     Enc/Outputs/Out/nCtrl1 <-> ENC Control compact/Control/Enable latch C
//     Enc/Outputs/Out/nCtrl1 @bit 3 <-> ENC Control compact/Control/Enable latch extern on negative edge
//     Enc/Outputs/Out/nCtrl1 @bit 1 <-> ENC Control compact/Control/Enable latch extern on positive edge
//     Enc/Outputs/Out/nCtrl1 @bit 2 <-> ENC Control compact/Control/Set counter
//     Enc/Outputs/Out/nDataOut1[0] <-> ENC Control compact/Set counter value
//   NC-Task 1 SAF/Axes/VGP_80 <-> =+-CX2020/EtherCAT1/=+-EK1100_04_00/=+-EL7041_04_04
//     Drive/Inputs/In/nState1 @bit 3 <-> STM Status/Status/Error
//     Drive/Inputs/In/nState1 @bit 5 <-> STM Status/Status/Moving negative
//     Drive/Inputs/In/nState1 @bit 4 <-> STM Status/Status/Moving positive
//     Drive/Inputs/In/nState1 @bit 1 <-> STM Status/Status/Ready
//     Drive/Inputs/In/nState1 <-> STM Status/Status/Ready to enable
//     Drive/Inputs/In/nState1 @bit 6 <-> STM Status/Status/Torque reduced
//     Drive/Inputs/In/nState1 @bit 2 <-> STM Status/Status/Warning
//     Drive/Inputs/In/nState2 @bit 3 <-> STM Status/Status/Digital input 1
//     Drive/Inputs/In/nState2 @bit 4 <-> STM Status/Status/Digital input 2
//     Drive/Inputs/In/nState2 @bit 5 <-> STM Status/Status/Sync error
//     Drive/Inputs/In/nState2 @bit 7 <-> STM Status/Status/TxPDO Toggle
//     Drive/Inputs/In/nState4 @bit 1 <-> WcState/InputToggle
//     Drive/Inputs/In/nState4 <-> WcState/WcState
//     Drive/Outputs/Out/nCtrl1 <-> STM Control/Control/Enable
//     Drive/Outputs/Out/nCtrl1 @bit 2 <-> STM Control/Control/Reduce torque
//     Drive/Outputs/Out/nCtrl1 @bit 1 <-> STM Control/Control/Reset
//     Drive/Outputs/Out/nDataOut2[0] <-> STM Velocity/Velocity
//   __THIS__ <-> plc_kfe_gatt/plc_kfe_gatt Instance
//     =+-EL2798_01_03/Channel 1/fb_AT1K0_GAS_GCC_10.q_xHV_DIS <-> PlcTask Outputs/GVL_Devices.fb_AT1K0_GAS_GCC_10.q_xHV_DIS
//     =+-EL2798_01_03/Channel 2/fb_AT1K0_GAS_GCC_20.q_xHV_DIS <-> PlcTask Outputs/GVL_Devices.fb_AT1K0_GAS_GCC_20.q_xHV_DIS
//     =+-EL2798_01_03/Channel 5/fb_AT1K0_GAS_GCC_30.q_xHV_DIS <-> PlcTask Outputs/GVL_Devices.fb_AT1K0_GAS_GCC_30.q_xHV_DIS
//     =+-EL2798_01_03/Channel 6/fb_AT1K0_GAS_GCC_40.q_xHV_DIS <-> PlcTask Outputs/GVL_Devices.fb_AT1K0_GAS_GCC_40.q_xHV_DIS
//     =+-EL2798_01_08/Channel 1/fb_AT1K0_GAS_GCC_50.q_xHV_DIS <-> PlcTask Outputs/GVL_Devices.fb_AT1K0_GAS_GCC_50.q_xHV_DIS
//     =+-EL2798_01_08/Channel 2/fb_AT1K0_GAS_GCC_60.q_xHV_DIS <-> PlcTask Outputs/GVL_Devices.fb_AT1K0_GAS_GCC_60.q_xHV_DIS
//     =+-EL2798_01_08/Channel 5/fb_AT1K0_GAS_GCC_80.q_xHV_DIS <-> PlcTask Outputs/GVL_Devices.fb_AT1K0_GAS_GCC_80.q_xHV_DIS
//     =+-EL2798_01_14/Channel 1/fb_AT1K0_GAS_GCC_90.q_xHV_DIS <-> PlcTask Outputs/GVL_Devices.fb_AT1K0_GAS_GCC_90.q_xHV_DIS
//     =+-EL2798_01_14/Channel 2/fb_AT1K0_GAS_GCC_100.q_xHV_DIS <-> PlcTask Outputs/GVL_Devices.fb_AT1K0_GAS_GCC_100.q_xHV_DIS
//     =+-EL2798_01_14/Channel 5/fb_AT1K0_GAS_GCC_110.q_xHV_DIS <-> PlcTask Outputs/GVL_Devices.fb_AT1K0_GAS_GCC_110.q_xHV_DIS
//     =+-EL2798_01_14/Channel 6/fb_AT1K0_GAS_GCC_120.q_xHV_DIS <-> PlcTask Outputs/GVL_Devices.fb_AT1K0_GAS_GCC_120.q_xHV_DIS
//     =+-EL2798_01_19/Channel 1/Output <-> PlcTask Outputs/GVL_Devices.fb_AT1K0_GAS_GCC_130.q_xHV_DIS
//     =+-EL2798_01_19/Channel 2/Output <-> PlcTask Outputs/GVL_Devices.fb_AT1K0_GAS_GCC_140.q_xHV_DIS
//     =+-ES3064_01_01/AI Standard Channel 1/fb_AT1K0_GAS_GCC_10.i_iPRESS_R <-> PlcTask Inputs/GVL_Devices.fb_AT1K0_GAS_GCC_10.i_iPRESS_R
//     =+-ES3064_01_01/AI Standard Channel 3/fb_AT1K0_GAS_GCC_20.i_iPRESS_R <-> PlcTask Inputs/GVL_Devices.fb_AT1K0_GAS_GCC_20.i_iPRESS_R
//     =+-ES3064_01_04/AI Standard Channel 1/fb_AT1K0_GAS_GCC_30.i_iPRESS_R <-> PlcTask Inputs/GVL_Devices.fb_AT1K0_GAS_GCC_30.i_iPRESS_R
//     =+-ES3064_01_04/AI Standard Channel 3/fb_AT1K0_GAS_GCC_40.i_iPRESS_R <-> PlcTask Inputs/GVL_Devices.fb_AT1K0_GAS_GCC_40.i_iPRESS_R
//     =+-ES3064_01_06/AI Standard Channel 1/fb_AT1K0_GAS_GCC_50.i_iPRESS_R <-> PlcTask Inputs/GVL_Devices.fb_AT1K0_GAS_GCC_50.i_iPRESS_R
//     =+-ES3064_01_06/AI Standard Channel 3/fb_AT1K0_GAS_GCC_60.i_iPRESS_R <-> PlcTask Inputs/GVL_Devices.fb_AT1K0_GAS_GCC_60.i_iPRESS_R
//     =+-ES3064_01_09/AI Standard Channel 1/fb_AT1K0_GAS_GCC_80.i_iPRESS_R <-> PlcTask Inputs/GVL_Devices.fb_AT1K0_GAS_GCC_80.i_iPRESS_R
//     =+-ES3064_01_12/AI Standard Channel 1/fb_AT1K0_GAS_GCC_90.i_iPRESS_R <-> PlcTask Inputs/GVL_Devices.fb_AT1K0_GAS_GCC_90.i_iPRESS_R
//     =+-ES3064_01_12/AI Standard Channel 3/fb_AT1K0_GAS_GCC_100.i_iPRESS_R <-> PlcTask Inputs/GVL_Devices.fb_AT1K0_GAS_GCC_100.i_iPRESS_R
//     =+-ES3064_01_15/AI Standard Channel 1/fb_AT1K0_GAS_GCC_110.i_iPRESS_R <-> PlcTask Inputs/GVL_Devices.fb_AT1K0_GAS_GCC_110.i_iPRESS_R
//     =+-ES3064_01_15/AI Standard Channel 3/fb_AT1K0_GAS_GCC_120.i_iPRESS_R <-> PlcTask Inputs/GVL_Devices.fb_AT1K0_GAS_GCC_120.i_iPRESS_R
//     =+-ES3064_01_17/AI Standard Channel 1/fb_AT1K0_GAS_GCC_130.i_iPRESS_R <-> PlcTask Inputs/GVL_Devices.fb_AT1K0_GAS_GCC_130.i_iPRESS_R
//     =+-ES3064_01_17/AI Standard Channel 3/fb_AT1K0_GAS_GCC_140.i_iPRESS_R <-> PlcTask Inputs/GVL_Devices.fb_AT1K0_GAS_GCC_140.i_iPRESS_R
//     =+-ES3064_01_02/AI Standard Channel 1/fb_AT1K0_GAS_GPI_10.i_iPRESS_R <-> PlcTask Inputs/GVL_Devices.fb_AT1K0_GAS_GPI_10.i_iPRESS_R
//     =+-ES3064_01_02/AI Standard Channel 2/fb_AT1K0_GAS_GPI_20.i_iPRESS_R <-> PlcTask Inputs/GVL_Devices.fb_AT1K0_GAS_GPI_20.i_iPRESS_R
//     =+-ES3064_01_05/AI Standard Channel 1/fb_AT1K0_GAS_GPI_30.i_iPRESS_R <-> PlcTask Inputs/GVL_Devices.fb_AT1K0_GAS_GPI_30.i_iPRESS_R
//     =+-ES3064_01_05/AI Standard Channel 2/fb_AT1K0_GAS_GPI_40.i_iPRESS_R <-> PlcTask Inputs/GVL_Devices.fb_AT1K0_GAS_GPI_40.i_iPRESS_R
//     =+-ES3064_01_07/AI Standard Channel 1/fb_AT1K0_GAS_GPI_50.i_iPRESS_R <-> PlcTask Inputs/GVL_Devices.fb_AT1K0_GAS_GPI_50.i_iPRESS_R
//     =+-ES3064_01_07/AI Standard Channel 2/fb_AT1K0_GAS_GPI_60.i_iPRESS_R <-> PlcTask Inputs/GVL_Devices.fb_AT1K0_GAS_GPI_60.i_iPRESS_R
//     =+-ES3064_01_09/AI Standard Channel 3/fb_AT1K0_GAS_GPI_80.i_iPRESS_R <-> PlcTask Inputs/GVL_Devices.fb_AT1K0_GAS_GPI_80.i_iPRESS_R
//     =+-ES3064_01_10/AI Standard Channel 1/fb_AT1K0_GAS_GPI_11.i_iPRESS_R <-> PlcTask Inputs/GVL_Devices.fb_AT1K0_GAS_GPI_11.i_iPRESS_R
//     =+-ES3064_01_10/AI Standard Channel 2/fb_AT1K0_GAS_GPI_51.i_iPRESS_R <-> PlcTask Inputs/GVL_Devices.fb_AT1K0_GAS_GPI_51.i_iPRESS_R
//     =+-ES3064_01_13/AI Standard Channel 1/fb_AT1K0_GAS_GPI_90.i_iPRESS_R <-> PlcTask Inputs/GVL_Devices.fb_AT1K0_GAS_GPI_90.i_iPRESS_R
//     =+-ES3064_01_13/AI Standard Channel 2/fb_AT1K0_GAS_GPI_100.i_iPRESS_R <-> PlcTask Inputs/GVL_Devices.fb_AT1K0_GAS_GPI_100.i_iPRESS_R
//     =+-ES3064_01_16/AI Standard Channel 1/fb_AT1K0_GAS_GPI_110.i_iPRESS_R <-> PlcTask Inputs/GVL_Devices.fb_AT1K0_GAS_GPI_110.i_iPRESS_R
//     =+-ES3064_01_16/AI Standard Channel 2/fb_AT1K0_GAS_GPI_120.i_iPRESS_R <-> PlcTask Inputs/GVL_Devices.fb_AT1K0_GAS_GPI_120.i_iPRESS_R
//     =+-ES3064_01_18/AI Standard Channel 1/fb_AT1K0_GAS_GPI_130.i_iPRESS_R <-> PlcTask Inputs/GVL_Devices.fb_AT1K0_GAS_GPI_130.i_iPRESS_R
//     =+-ES3064_01_18/AI Standard Channel 2/fb_AT1K0_GAS_GPI_140.i_iPRESS_R <-> PlcTask Inputs/GVL_Devices.fb_AT1K0_GAS_GPI_140.i_iPRESS_R
//     =+-EL2798_03_03/Channel 1/fb_AT1K0_GAS_PTM_10.q_xReset <-> PlcTask Outputs/GVL_Devices.fb_AT1K0_GAS_PTM_10.q_xReset
//     =+-EL2798_03_07/Channel 1/fb_AT1K0_GAS_PTM_20.q_xReset <-> PlcTask Outputs/GVL_Devices.fb_AT1K0_GAS_PTM_20.q_xReset
//     =+-EL2798_03_13/Channel 1/fb_AT1K0_GAS_PTM_30.q_xReset <-> PlcTask Outputs/GVL_Devices.fb_AT1K0_GAS_PTM_30.q_xReset
//     =+-EL2798_03_17/Channel 1/fb_AT1K0_GAS_PTM_40.q_xReset <-> PlcTask Outputs/GVL_Devices.fb_AT1K0_GAS_PTM_40.q_xReset
//     =+-EL2798_03_03/Channel 2/fb_AT1K0_GAS_PTM_10.q_xStart <-> PlcTask Outputs/GVL_Devices.fb_AT1K0_GAS_PTM_10.q_xStart
//     =+-EL2798_03_07/Channel 2/fb_AT1K0_GAS_PTM_20.q_xStart <-> PlcTask Outputs/GVL_Devices.fb_AT1K0_GAS_PTM_20.q_xStart
//     =+-EL2798_03_13/Channel 2/fb_AT1K0_GAS_PTM_30.q_xStart <-> PlcTask Outputs/GVL_Devices.fb_AT1K0_GAS_PTM_30.q_xStart
//     =+-EL2798_03_17/Channel 2/fb_AT1K0_GAS_PTM_40.q_xStart <-> PlcTask Outputs/GVL_Devices.fb_AT1K0_GAS_PTM_40.q_xStart
//     =+-EL2798_03_03/Channel 3/fb_AT1K0_GAS_PTM_10.q_xStop <-> PlcTask Outputs/GVL_Devices.fb_AT1K0_GAS_PTM_10.q_xStop
//     =+-EL2798_03_07/Channel 3/fb_AT1K0_GAS_PTM_20.q_xStop <-> PlcTask Outputs/GVL_Devices.fb_AT1K0_GAS_PTM_20.q_xStop
//     =+-EL2798_03_13/Channel 3/fb_AT1K0_GAS_PTM_30.q_xStop <-> PlcTask Outputs/GVL_Devices.fb_AT1K0_GAS_PTM_30.q_xStop
//     =+-EL2798_03_17/Channel 3/fb_AT1K0_GAS_PTM_40.q_xStop <-> PlcTask Outputs/GVL_Devices.fb_AT1K0_GAS_PTM_40.q_xStop
//     =+-EL2798_03_03/Channel 4/fb_AT1K0_GAS_PTM_10.q_xProtection <-> PlcTask Outputs/GVL_Devices.fb_AT1K0_GAS_PTM_10.q_xProtection
//     =+-EL2798_03_07/Channel 4/fb_AT1K0_GAS_PTM_20.q_xProtection <-> PlcTask Outputs/GVL_Devices.fb_AT1K0_GAS_PTM_20.q_xProtection
//     =+-EL2798_03_13/Channel 4/fb_AT1K0_GAS_PTM_30.q_xProtection <-> PlcTask Outputs/GVL_Devices.fb_AT1K0_GAS_PTM_30.q_xProtection
//     =+-EL2798_03_17/Channel 4/fb_AT1K0_GAS_PTM_40.q_xProtection <-> PlcTask Outputs/GVL_Devices.fb_AT1K0_GAS_PTM_40.q_xProtection
//     =+-EL2798_03_03/Channel 5/fb_AT1K0_GAS_PTM_10.q_xSetSpeed <-> PlcTask Outputs/GVL_Devices.fb_AT1K0_GAS_PTM_10.q_xSetSpeed
//     =+-EL2798_03_07/Channel 5/fb_AT1K0_GAS_PTM_20.q_xSetSpeed <-> PlcTask Outputs/GVL_Devices.fb_AT1K0_GAS_PTM_20.q_xSetSpeed
//     =+-EL2798_03_13/Channel 5/fb_AT1K0_GAS_PTM_30.q_xSetSpeed <-> PlcTask Outputs/GVL_Devices.fb_AT1K0_GAS_PTM_30.q_xSetSpeed
//     =+-EL2798_03_17/Channel 5/fb_AT1K0_GAS_PTM_40.q_xSetSpeed <-> PlcTask Outputs/GVL_Devices.fb_AT1K0_GAS_PTM_40.q_xSetSpeed
//     =+-ES1004_03_01/Channel 1/fb_AT1K0_GAS_PTM_10.i_xDecel <-> PlcTask Inputs/GVL_Devices.fb_AT1K0_GAS_PTM_10.i_xDecel
//     =+-ES1004_03_08/Channel 1/fb_AT1K0_GAS_PTM_20.i_xDecel <-> PlcTask Inputs/GVL_Devices.fb_AT1K0_GAS_PTM_20.i_xDecel
//     =+-ES1004_03_11/Channel 1/fb_AT1K0_GAS_PTM_30.i_xDecel <-> PlcTask Inputs/GVL_Devices.fb_AT1K0_GAS_PTM_30.i_xDecel
//     =+-ES1004_03_18/Channel 1/fb_AT1K0_GAS_PTM_40.i_xDecel <-> PlcTask Inputs/GVL_Devices.fb_AT1K0_GAS_PTM_40.i_xDecel
//     =+-ES1004_03_01/Channel 2/fb_AT1K0_GAS_PTM_10.i_xAtSpd <-> PlcTask Inputs/GVL_Devices.fb_AT1K0_GAS_PTM_10.i_xAtSpd
//     =+-ES1004_03_08/Channel 2/fb_AT1K0_GAS_PTM_20.i_xAtSpd <-> PlcTask Inputs/GVL_Devices.fb_AT1K0_GAS_PTM_20.i_xAtSpd
//     =+-ES1004_03_11/Channel 2/fb_AT1K0_GAS_PTM_30.i_xAtSpd <-> PlcTask Inputs/GVL_Devices.fb_AT1K0_GAS_PTM_30.i_xAtSpd
//     =+-ES1004_03_18/Channel 2/fb_AT1K0_GAS_PTM_40.i_xAtSpd <-> PlcTask Inputs/GVL_Devices.fb_AT1K0_GAS_PTM_40.i_xAtSpd
//     =+-ES1004_03_01/Channel 3/fb_AT1K0_GAS_PTM_10.i_xNCFault <-> PlcTask Inputs/GVL_Devices.fb_AT1K0_GAS_PTM_10.i_xNCFault
//     =+-ES1004_03_08/Channel 3/fb_AT1K0_GAS_PTM_20.i_xNCFault <-> PlcTask Inputs/GVL_Devices.fb_AT1K0_GAS_PTM_20.i_xNCFault
//     =+-ES1004_03_11/Channel 3/fb_AT1K0_GAS_PTM_30.i_xNCFault <-> PlcTask Inputs/GVL_Devices.fb_AT1K0_GAS_PTM_30.i_xNCFault
//     =+-ES1004_03_18/Channel 3/fb_AT1K0_GAS_PTM_40.i_xNCFault <-> PlcTask Inputs/GVL_Devices.fb_AT1K0_GAS_PTM_40.i_xNCFault
//     =+-ES1004_03_01/Channel 4/fb_AT1K0_GAS_PTM_10.i_xRotate <-> PlcTask Inputs/GVL_Devices.fb_AT1K0_GAS_PTM_10.i_xRotate
//     =+-ES1004_03_08/Channel 4/fb_AT1K0_GAS_PTM_20.i_xRotate <-> PlcTask Inputs/GVL_Devices.fb_AT1K0_GAS_PTM_20.i_xRotate
//     =+-ES1004_03_11/Channel 4/fb_AT1K0_GAS_PTM_30.i_xRotate <-> PlcTask Inputs/GVL_Devices.fb_AT1K0_GAS_PTM_30.i_xRotate
//     =+-ES1004_03_18/Channel 4/fb_AT1K0_GAS_PTM_40.i_xRotate <-> PlcTask Inputs/GVL_Devices.fb_AT1K0_GAS_PTM_40.i_xRotate
//     =+-ES1004_03_02/Channel 1/fb_AT1K0_GAS_PTM_10.i_xAccel <-> PlcTask Inputs/GVL_Devices.fb_AT1K0_GAS_PTM_10.i_xAccel
//     =+-ES1004_03_09/Channel 1/fb_AT1K0_GAS_PTM_20.i_xAccel <-> PlcTask Inputs/GVL_Devices.fb_AT1K0_GAS_PTM_20.i_xAccel
//     =+-ES1004_03_12/Channel 1/fb_AT1K0_GAS_PTM_30.i_xAccel <-> PlcTask Inputs/GVL_Devices.fb_AT1K0_GAS_PTM_30.i_xAccel
//     =+-ES1004_03_19/Channel 1/fb_AT1K0_GAS_PTM_40.i_xAccel <-> PlcTask Inputs/GVL_Devices.fb_AT1K0_GAS_PTM_40.i_xAccel
//     =+-ES3064_03_04/AI Standard Channel 1/fb_AT1K0_GAS_PTM_10.i_iRawSpeed <-> PlcTask Inputs/GVL_Devices.fb_AT1K0_GAS_PTM_10.i_iRawSpeed
//     =+-ES3064_03_06/AI Standard Channel 1/fb_AT1K0_GAS_PTM_20.i_iRawSpeed <-> PlcTask Inputs/GVL_Devices.fb_AT1K0_GAS_PTM_20.i_iRawSpeed
//     =+-ES3064_03_14/AI Standard Channel 1/fb_AT1K0_GAS_PTM_30.i_iRawSpeed <-> PlcTask Inputs/GVL_Devices.fb_AT1K0_GAS_PTM_30.i_iRawSpeed
//     =+-ES3064_03_16/AI Standard Channel 1/fb_AT1K0_GAS_PTM_40.i_iRawSpeed <-> PlcTask Inputs/GVL_Devices.fb_AT1K0_GAS_PTM_40.i_iRawSpeed
//     =+-ES3064_03_04/AI Standard Channel 2/fb_AT1K0_GAS_PTM_10.i_iCurrentMon <-> PlcTask Inputs/GVL_Devices.fb_AT1K0_GAS_PTM_10.i_iCurrentMon
//     =+-ES3064_03_06/AI Standard Channel 2/fb_AT1K0_GAS_PTM_20.i_iCurrentMon <-> PlcTask Inputs/GVL_Devices.fb_AT1K0_GAS_PTM_20.i_iCurrentMon
//     =+-ES3064_03_14/AI Standard Channel 2/fb_AT1K0_GAS_PTM_30.i_iCurrentMon <-> PlcTask Inputs/GVL_Devices.fb_AT1K0_GAS_PTM_30.i_iCurrentMon
//     =+-ES3064_03_16/AI Standard Channel 2/fb_AT1K0_GAS_PTM_40.i_iCurrentMon <-> PlcTask Inputs/GVL_Devices.fb_AT1K0_GAS_PTM_40.i_iCurrentMon
//     =+-ES3064_03_04/AI Standard Channel 3/fb_AT1K0_GAS_PTM_10.i_iTempMon <-> PlcTask Inputs/GVL_Devices.fb_AT1K0_GAS_PTM_10.i_iTempMon
//     =+-ES3064_03_06/AI Standard Channel 3/fb_AT1K0_GAS_PTM_20.i_iTempMon <-> PlcTask Inputs/GVL_Devices.fb_AT1K0_GAS_PTM_20.i_iTempMon
//     =+-ES3064_03_14/AI Standard Channel 3/fb_AT1K0_GAS_PTM_30.i_iTempMon <-> PlcTask Inputs/GVL_Devices.fb_AT1K0_GAS_PTM_30.i_iTempMon
//     =+-ES3064_03_16/AI Standard Channel 3/fb_AT1K0_GAS_PTM_40.i_iTempMon <-> PlcTask Inputs/GVL_Devices.fb_AT1K0_GAS_PTM_40.i_iTempMon
//     =+-ES4004_03_05/AO Outputs Channel 1/fb_AT1K0_GAS_PTM_10.q_iSpeedSet <-> PlcTask Outputs/GVL_Devices.fb_AT1K0_GAS_PTM_10.q_iSpeedSet
//     =+-ES4004_03_05/AO Outputs Channel 3/fb_AT1K0_GAS_PTM_20.q_iSpeedSet <-> PlcTask Outputs/GVL_Devices.fb_AT1K0_GAS_PTM_20.q_iSpeedSet
//     =+-ES4004_03_15/AO Outputs Channel 1/fb_AT1K0_GAS_PTM_30.q_iSpeedSet <-> PlcTask Outputs/GVL_Devices.fb_AT1K0_GAS_PTM_30.q_iSpeedSet
//     =+-ES4004_03_15/AO Outputs Channel 3/fb_AT1K0_GAS_PTM_40.q_iSpeedSet <-> PlcTask Outputs/GVL_Devices.fb_AT1K0_GAS_PTM_40.q_iSpeedSet
//   plc_kfe_gatt Instance <-> =+-CX2020/EtherCAT1
//     PlcTask Inputs/DIAGNOSTICS.i_sAMSNetID <-> InfoData/AmsNetId
//     PlcTask Inputs/GVL_GATT.fbEcatDiagWrapper.nEcMasterDevState <-> Inputs/DevState
//     PlcTask Inputs/GVL_GATT.fbEcatDiagWrapper.nEcMasterDeviceId <-> InfoData/DevId
//     PlcTask Inputs/GVL_GATT.fbEcatDiagWrapper.nEcMasterSlaveCount <-> Inputs/SlaveCount
//   plc_kfe_gatt Instance <-> =+-CX2020/EtherCAT1/=+-EK1100_01_00/=+-EL2798_01_03
//     PlcTask Outputs/GVL_Devices.fb_AT1K0_GAS_GCC_10.q_xHV_DIS <-> Channel 1/fb_AT1K0_GAS_GCC_10.q_xHV_DIS
//     PlcTask Outputs/GVL_Devices.fb_AT1K0_GAS_GCC_20.q_xHV_DIS <-> Channel 2/fb_AT1K0_GAS_GCC_20.q_xHV_DIS
//     PlcTask Outputs/GVL_Devices.fb_AT1K0_GAS_GCC_30.q_xHV_DIS <-> Channel 5/fb_AT1K0_GAS_GCC_30.q_xHV_DIS
//     PlcTask Outputs/GVL_Devices.fb_AT1K0_GAS_GCC_40.q_xHV_DIS <-> Channel 6/fb_AT1K0_GAS_GCC_40.q_xHV_DIS
//   plc_kfe_gatt Instance <-> =+-CX2020/EtherCAT1/=+-EK1100_01_00/=+-EL2798_01_08
//     PlcTask Outputs/GVL_Devices.fb_AT1K0_GAS_GCC_50.q_xHV_DIS <-> Channel 1/fb_AT1K0_GAS_GCC_50.q_xHV_DIS
//     PlcTask Outputs/GVL_Devices.fb_AT1K0_GAS_GCC_60.q_xHV_DIS <-> Channel 2/fb_AT1K0_GAS_GCC_60.q_xHV_DIS
//     PlcTask Outputs/GVL_Devices.fb_AT1K0_GAS_GCC_80.q_xHV_DIS <-> Channel 5/fb_AT1K0_GAS_GCC_80.q_xHV_DIS
//   plc_kfe_gatt Instance <-> =+-CX2020/EtherCAT1/=+-EK1100_01_00/=+-EL2798_01_14
//     PlcTask Outputs/GVL_Devices.fb_AT1K0_GAS_GCC_100.q_xHV_DIS <-> Channel 2/fb_AT1K0_GAS_GCC_100.q_xHV_DIS
//     PlcTask Outputs/GVL_Devices.fb_AT1K0_GAS_GCC_110.q_xHV_DIS <-> Channel 5/fb_AT1K0_GAS_GCC_110.q_xHV_DIS
//     PlcTask Outputs/GVL_Devices.fb_AT1K0_GAS_GCC_120.q_xHV_DIS <-> Channel 6/fb_AT1K0_GAS_GCC_120.q_xHV_DIS
//     PlcTask Outputs/GVL_Devices.fb_AT1K0_GAS_GCC_90.q_xHV_DIS <-> Channel 1/fb_AT1K0_GAS_GCC_90.q_xHV_DIS
//   plc_kfe_gatt Instance <-> =+-CX2020/EtherCAT1/=+-EK1100_01_00/=+-EL2798_01_19
//     PlcTask Outputs/GVL_Devices.fb_AT1K0_GAS_GCC_130.q_xHV_DIS <-> Channel 1/Output
//     PlcTask Outputs/GVL_Devices.fb_AT1K0_GAS_GCC_140.q_xHV_DIS <-> Channel 2/Output
//   plc_kfe_gatt Instance <-> =+-CX2020/EtherCAT1/=+-EK1100_01_00/=+-ES3064_01_01
//     PlcTask Inputs/GVL_Devices.fb_AT1K0_GAS_GCC_10.i_iPRESS_R <-> AI Standard Channel 1/fb_AT1K0_GAS_GCC_10.i_iPRESS_R
//     PlcTask Inputs/GVL_Devices.fb_AT1K0_GAS_GCC_20.i_iPRESS_R <-> AI Standard Channel 3/fb_AT1K0_GAS_GCC_20.i_iPRESS_R
//   plc_kfe_gatt Instance <-> =+-CX2020/EtherCAT1/=+-EK1100_01_00/=+-ES3064_01_02
//     PlcTask Inputs/GVL_Devices.fb_AT1K0_GAS_GPI_10.i_iPRESS_R <-> AI Standard Channel 1/fb_AT1K0_GAS_GPI_10.i_iPRESS_R
//     PlcTask Inputs/GVL_Devices.fb_AT1K0_GAS_GPI_20.i_iPRESS_R <-> AI Standard Channel 2/fb_AT1K0_GAS_GPI_20.i_iPRESS_R
//   plc_kfe_gatt Instance <-> =+-CX2020/EtherCAT1/=+-EK1100_01_00/=+-ES3064_01_04
//     PlcTask Inputs/GVL_Devices.fb_AT1K0_GAS_GCC_30.i_iPRESS_R <-> AI Standard Channel 1/fb_AT1K0_GAS_GCC_30.i_iPRESS_R
//     PlcTask Inputs/GVL_Devices.fb_AT1K0_GAS_GCC_40.i_iPRESS_R <-> AI Standard Channel 3/fb_AT1K0_GAS_GCC_40.i_iPRESS_R
//   plc_kfe_gatt Instance <-> =+-CX2020/EtherCAT1/=+-EK1100_01_00/=+-ES3064_01_05
//     PlcTask Inputs/GVL_Devices.fb_AT1K0_GAS_GPI_30.i_iPRESS_R <-> AI Standard Channel 1/fb_AT1K0_GAS_GPI_30.i_iPRESS_R
//     PlcTask Inputs/GVL_Devices.fb_AT1K0_GAS_GPI_40.i_iPRESS_R <-> AI Standard Channel 2/fb_AT1K0_GAS_GPI_40.i_iPRESS_R
//   plc_kfe_gatt Instance <-> =+-CX2020/EtherCAT1/=+-EK1100_01_00/=+-ES3064_01_06
//     PlcTask Inputs/GVL_Devices.fb_AT1K0_GAS_GCC_50.i_iPRESS_R <-> AI Standard Channel 1/fb_AT1K0_GAS_GCC_50.i_iPRESS_R
//     PlcTask Inputs/GVL_Devices.fb_AT1K0_GAS_GCC_60.i_iPRESS_R <-> AI Standard Channel 3/fb_AT1K0_GAS_GCC_60.i_iPRESS_R
//   plc_kfe_gatt Instance <-> =+-CX2020/EtherCAT1/=+-EK1100_01_00/=+-ES3064_01_07
//     PlcTask Inputs/GVL_Devices.fb_AT1K0_GAS_GPI_50.i_iPRESS_R <-> AI Standard Channel 1/fb_AT1K0_GAS_GPI_50.i_iPRESS_R
//     PlcTask Inputs/GVL_Devices.fb_AT1K0_GAS_GPI_60.i_iPRESS_R <-> AI Standard Channel 2/fb_AT1K0_GAS_GPI_60.i_iPRESS_R
//   plc_kfe_gatt Instance <-> =+-CX2020/EtherCAT1/=+-EK1100_01_00/=+-ES3064_01_09
//     PlcTask Inputs/GVL_Devices.fb_AT1K0_GAS_GCC_80.i_iPRESS_R <-> AI Standard Channel 1/fb_AT1K0_GAS_GCC_80.i_iPRESS_R
//     PlcTask Inputs/GVL_Devices.fb_AT1K0_GAS_GPI_12.i_iPRESS_R <-> AI Standard Channel 4/Value
//     PlcTask Inputs/GVL_Devices.fb_AT1K0_GAS_GPI_80.i_iPRESS_R <-> AI Standard Channel 3/fb_AT1K0_GAS_GPI_80.i_iPRESS_R
//   plc_kfe_gatt Instance <-> =+-CX2020/EtherCAT1/=+-EK1100_01_00/=+-ES3064_01_10
//     PlcTask Inputs/GVL_Devices.fb_AT1K0_GAS_GPI_11.i_iPRESS_R <-> AI Standard Channel 1/fb_AT1K0_GAS_GPI_11.i_iPRESS_R
//     PlcTask Inputs/GVL_Devices.fb_AT1K0_GAS_GPI_51.i_iPRESS_R <-> AI Standard Channel 2/fb_AT1K0_GAS_GPI_51.i_iPRESS_R
//   plc_kfe_gatt Instance <-> =+-CX2020/EtherCAT1/=+-EK1100_01_00/=+-ES3064_01_12
//     PlcTask Inputs/GVL_Devices.fb_AT1K0_GAS_GCC_100.i_iPRESS_R <-> AI Standard Channel 3/fb_AT1K0_GAS_GCC_100.i_iPRESS_R
//     PlcTask Inputs/GVL_Devices.fb_AT1K0_GAS_GCC_90.i_iPRESS_R <-> AI Standard Channel 1/fb_AT1K0_GAS_GCC_90.i_iPRESS_R
//   plc_kfe_gatt Instance <-> =+-CX2020/EtherCAT1/=+-EK1100_01_00/=+-ES3064_01_13
//     PlcTask Inputs/GVL_Devices.fb_AT1K0_GAS_GPI_100.i_iPRESS_R <-> AI Standard Channel 2/fb_AT1K0_GAS_GPI_100.i_iPRESS_R
//     PlcTask Inputs/GVL_Devices.fb_AT1K0_GAS_GPI_90.i_iPRESS_R <-> AI Standard Channel 1/fb_AT1K0_GAS_GPI_90.i_iPRESS_R
//   plc_kfe_gatt Instance <-> =+-CX2020/EtherCAT1/=+-EK1100_01_00/=+-ES3064_01_15
//     PlcTask Inputs/GVL_Devices.fb_AT1K0_GAS_GCC_110.i_iPRESS_R <-> AI Standard Channel 1/fb_AT1K0_GAS_GCC_110.i_iPRESS_R
//     PlcTask Inputs/GVL_Devices.fb_AT1K0_GAS_GCC_120.i_iPRESS_R <-> AI Standard Channel 3/fb_AT1K0_GAS_GCC_120.i_iPRESS_R
//   plc_kfe_gatt Instance <-> =+-CX2020/EtherCAT1/=+-EK1100_01_00/=+-ES3064_01_16
//     PlcTask Inputs/GVL_Devices.fb_AT1K0_GAS_GPI_110.i_iPRESS_R <-> AI Standard Channel 1/fb_AT1K0_GAS_GPI_110.i_iPRESS_R
//     PlcTask Inputs/GVL_Devices.fb_AT1K0_GAS_GPI_120.i_iPRESS_R <-> AI Standard Channel 2/fb_AT1K0_GAS_GPI_120.i_iPRESS_R
//   plc_kfe_gatt Instance <-> =+-CX2020/EtherCAT1/=+-EK1100_01_00/=+-ES3064_01_17
//     PlcTask Inputs/GVL_Devices.fb_AT1K0_GAS_GCC_130.i_iPRESS_R <-> AI Standard Channel 1/fb_AT1K0_GAS_GCC_130.i_iPRESS_R
//     PlcTask Inputs/GVL_Devices.fb_AT1K0_GAS_GCC_140.i_iPRESS_R <-> AI Standard Channel 3/fb_AT1K0_GAS_GCC_140.i_iPRESS_R
//   plc_kfe_gatt Instance <-> =+-CX2020/EtherCAT1/=+-EK1100_01_00/=+-ES3064_01_18
//     PlcTask Inputs/GVL_Devices.fb_AT1K0_GAS_GPI_130.i_iPRESS_R <-> AI Standard Channel 1/fb_AT1K0_GAS_GPI_130.i_iPRESS_R
//     PlcTask Inputs/GVL_Devices.fb_AT1K0_GAS_GPI_140.i_iPRESS_R <-> AI Standard Channel 2/fb_AT1K0_GAS_GPI_140.i_iPRESS_R
//   plc_kfe_gatt Instance <-> =+-CX2020/EtherCAT1/=+-EK1100_02_00/=+-ES1004_02_02
//     PlcTask Inputs/GVL_Devices.fb_AT1K0_GAS_VRC_10.i_xClsLS <-> Channel 2/fb_AT1K0_GAS_VRC_10.i_xClsLS
//     PlcTask Inputs/GVL_Devices.fb_AT1K0_GAS_VRC_20.i_xClsLS <-> Channel 4/fb_AT1K0_GAS_VRC_20.i_xClsLS
//     PlcTask Inputs/GVL_Devices.fb_AT1K0_GAS_VRC_10.i_xOpnLS <-> Channel 1/fb_AT1K0_GAS_VRC_10.i_xOpnLS
//     PlcTask Inputs/GVL_Devices.fb_AT1K0_GAS_VRC_20.i_xOpnLS <-> Channel 3/fb_AT1K0_GAS_VRC_20.i_xOpnLS
//   plc_kfe_gatt Instance <-> =+-CX2020/EtherCAT1/=+-EK1100_02_00/=+-ES1004_02_04
//     PlcTask Inputs/GVL_Devices.fb_AT1K0_GAS_VRC_30.i_xClsLS <-> Channel 2/fb_AT1K0_GAS_VRC_30.i_xClsLS
//     PlcTask Inputs/GVL_Devices.fb_AT1K0_GAS_VRC_40.i_xClsLS <-> Channel 4/fb_AT1K0_GAS_VRC_40.i_xClsLS
//     PlcTask Inputs/GVL_Devices.fb_AT1K0_GAS_VRC_30.i_xOpnLS <-> Channel 1/fb_AT1K0_GAS_VRC_30.i_xOpnLS
//     PlcTask Inputs/GVL_Devices.fb_AT1K0_GAS_VRC_40.i_xOpnLS <-> Channel 3/fb_AT1K0_GAS_VRC_40.i_xOpnLS
//   plc_kfe_gatt Instance <-> =+-CX2020/EtherCAT1/=+-EK1100_02_00/=+-ES1004_02_08
//     PlcTask Inputs/GVL_Devices.fb_AT1K0_GAS_VRC_50.i_xClsLS <-> Channel 2/Input
//     PlcTask Inputs/GVL_Devices.fb_AT1K0_GAS_VRC_60.i_xClsLS <-> Channel 4/Input
//     PlcTask Inputs/GVL_Devices.fb_AT1K0_GAS_VRC_50.i_xOpnLS <-> Channel 1/Input
//     PlcTask Inputs/GVL_Devices.fb_AT1K0_GAS_VRC_60.i_xOpnLS <-> Channel 3/Input
//   plc_kfe_gatt Instance <-> =+-CX2020/EtherCAT1/=+-EK1100_02_00/=+-ES2004_02_01
//     PlcTask Outputs/GVL_Devices.fb_AT1K0_GAS_VRC_10.q_xOPN_DO <-> Channel 1/fb_AT1K0_GAS_VRC_10.q_xOPN_DO
//     PlcTask Outputs/GVL_Devices.fb_AT1K0_GAS_VRC_20.q_xOPN_DO <-> Channel 3/fb_AT1K0_GAS_VRC_20.q_xOPN_DO
//     PlcTask Outputs/GVL_Devices.fb_AT1K0_GAS_VRC_10.q_xOPN_DO_2 <-> Channel 2/fb_AT1K0_GAS_VRC_10.q_xOPN_DO
//     PlcTask Outputs/GVL_Devices.fb_AT1K0_GAS_VRC_20.q_xOPN_DO_2 <-> Channel 4/fb_AT1K0_GAS_VRC_20.q_xOPN_DO
//   plc_kfe_gatt Instance <-> =+-CX2020/EtherCAT1/=+-EK1100_02_00/=+-ES2004_02_03
//     PlcTask Outputs/GVL_Devices.fb_AT1K0_GAS_VRC_30.q_xOPN_DO <-> Channel 1/fb_AT1K0_GAS_VRC_30.q_xOPN_DO
//     PlcTask Outputs/GVL_Devices.fb_AT1K0_GAS_VRC_40.q_xOPN_DO <-> Channel 3/fb_AT1K0_GAS_VRC_40.q_xOPN_DO
//     PlcTask Outputs/GVL_Devices.fb_AT1K0_GAS_VRC_30.q_xOPN_DO_2 <-> Channel 2/fb_AT1K0_GAS_VRC_30.q_xOPN_DO
//     PlcTask Outputs/GVL_Devices.fb_AT1K0_GAS_VRC_40.q_xOPN_DO_2 <-> Channel 4/fb_AT1K0_GAS_VRC_40.q_xOPN_DO
//   plc_kfe_gatt Instance <-> =+-CX2020/EtherCAT1/=+-EK1100_02_00/=+-ES2004_02_07
//     PlcTask Outputs/GVL_Devices.fb_AT1K0_GAS_VRC_50.q_xOPN_DO <-> Channel 1/Output
//     PlcTask Outputs/GVL_Devices.fb_AT1K0_GAS_VRC_60.q_xOPN_DO <-> Channel 2/Output
//     PlcTask Outputs/Main.M2.bBrakeRelease <-> Channel 3/Output
//     PlcTask Outputs/Main.M4.bBrakeRelease <-> Channel 4/Output
//   plc_kfe_gatt Instance <-> =+-CX2020/EtherCAT1/=+-EK1100_02_00/=+-ES2008_02_14
//     PlcTask Outputs/GVL_Devices.fb_AT1K0_GAS_VRC_11.q_xOPN_DO <-> Channel 1/Output
//   plc_kfe_gatt Instance <-> =+-CX2020/EtherCAT1/=+-EK1100_02_00/=+-ES7041_02_05
//     PlcTask Inputs/Main.M1.bLimitBackwardEnable <-> STM Status/Status/Digital input 2
//     PlcTask Inputs/Main.M1.bLimitForwardEnable <-> STM Status/Status/Digital input 1
//   plc_kfe_gatt Instance <-> =+-CX2020/EtherCAT1/=+-EK1100_02_00/=+-ES7041_02_06
//     PlcTask Inputs/Main.M2.bLimitBackwardEnable <-> STM Status/Status/Digital input 1
//     PlcTask Inputs/Main.M2.bLimitForwardEnable <-> STM Status/Status/Digital input 2
//   plc_kfe_gatt Instance <-> =+-CX2020/EtherCAT1/=+-EK1100_02_00/=+-ES7041_02_09
//     PlcTask Inputs/Main.M3.bLimitBackwardEnable <-> STM Status/Status/Digital input 2
//     PlcTask Inputs/Main.M3.bLimitForwardEnable <-> STM Status/Status/Digital input 1
//   plc_kfe_gatt Instance <-> =+-CX2020/EtherCAT1/=+-EK1100_02_00/=+-ES7041_02_10
//     PlcTask Inputs/Main.M4.bLimitBackwardEnable <-> STM Status/Status/Digital input 1
//     PlcTask Inputs/Main.M4.bLimitForwardEnable <-> STM Status/Status/Digital input 2
//   plc_kfe_gatt Instance <-> =+-CX2020/EtherCAT1/=+-EK1100_03_00/=+-EL2798_03_03
//     PlcTask Outputs/GVL_Devices.fb_AT1K0_GAS_PTM_10.q_xProtection <-> Channel 4/fb_AT1K0_GAS_PTM_10.q_xProtection
//     PlcTask Outputs/GVL_Devices.fb_AT1K0_GAS_PTM_10.q_xReset <-> Channel 1/fb_AT1K0_GAS_PTM_10.q_xReset
//     PlcTask Outputs/GVL_Devices.fb_AT1K0_GAS_PTM_10.q_xSetSpeed <-> Channel 5/fb_AT1K0_GAS_PTM_10.q_xSetSpeed
//     PlcTask Outputs/GVL_Devices.fb_AT1K0_GAS_PTM_10.q_xStart <-> Channel 2/fb_AT1K0_GAS_PTM_10.q_xStart
//     PlcTask Outputs/GVL_Devices.fb_AT1K0_GAS_PTM_10.q_xStop <-> Channel 3/fb_AT1K0_GAS_PTM_10.q_xStop
//   plc_kfe_gatt Instance <-> =+-CX2020/EtherCAT1/=+-EK1100_03_00/=+-EL2798_03_07
//     PlcTask Outputs/GVL_Devices.fb_AT1K0_GAS_PTM_20.q_xProtection <-> Channel 4/fb_AT1K0_GAS_PTM_20.q_xProtection
//     PlcTask Outputs/GVL_Devices.fb_AT1K0_GAS_PTM_20.q_xReset <-> Channel 1/fb_AT1K0_GAS_PTM_20.q_xReset
//     PlcTask Outputs/GVL_Devices.fb_AT1K0_GAS_PTM_20.q_xSetSpeed <-> Channel 5/fb_AT1K0_GAS_PTM_20.q_xSetSpeed
//     PlcTask Outputs/GVL_Devices.fb_AT1K0_GAS_PTM_20.q_xStart <-> Channel 2/fb_AT1K0_GAS_PTM_20.q_xStart
//     PlcTask Outputs/GVL_Devices.fb_AT1K0_GAS_PTM_20.q_xStop <-> Channel 3/fb_AT1K0_GAS_PTM_20.q_xStop
//   plc_kfe_gatt Instance <-> =+-CX2020/EtherCAT1/=+-EK1100_03_00/=+-EL2798_03_13
//     PlcTask Outputs/GVL_Devices.fb_AT1K0_GAS_PTM_30.q_xProtection <-> Channel 4/fb_AT1K0_GAS_PTM_30.q_xProtection
//     PlcTask Outputs/GVL_Devices.fb_AT1K0_GAS_PTM_30.q_xReset <-> Channel 1/fb_AT1K0_GAS_PTM_30.q_xReset
//     PlcTask Outputs/GVL_Devices.fb_AT1K0_GAS_PTM_30.q_xSetSpeed <-> Channel 5/fb_AT1K0_GAS_PTM_30.q_xSetSpeed
//     PlcTask Outputs/GVL_Devices.fb_AT1K0_GAS_PTM_30.q_xStart <-> Channel 2/fb_AT1K0_GAS_PTM_30.q_xStart
//     PlcTask Outputs/GVL_Devices.fb_AT1K0_GAS_PTM_30.q_xStop <-> Channel 3/fb_AT1K0_GAS_PTM_30.q_xStop
//   plc_kfe_gatt Instance <-> =+-CX2020/EtherCAT1/=+-EK1100_03_00/=+-EL2798_03_17
//     PlcTask Outputs/GVL_Devices.fb_AT1K0_GAS_PTM_40.q_xProtection <-> Channel 4/fb_AT1K0_GAS_PTM_40.q_xProtection
//     PlcTask Outputs/GVL_Devices.fb_AT1K0_GAS_PTM_40.q_xReset <-> Channel 1/fb_AT1K0_GAS_PTM_40.q_xReset
//     PlcTask Outputs/GVL_Devices.fb_AT1K0_GAS_PTM_40.q_xSetSpeed <-> Channel 5/fb_AT1K0_GAS_PTM_40.q_xSetSpeed
//     PlcTask Outputs/GVL_Devices.fb_AT1K0_GAS_PTM_40.q_xStart <-> Channel 2/fb_AT1K0_GAS_PTM_40.q_xStart
//     PlcTask Outputs/GVL_Devices.fb_AT1K0_GAS_PTM_40.q_xStop <-> Channel 3/fb_AT1K0_GAS_PTM_40.q_xStop
//   plc_kfe_gatt Instance <-> =+-CX2020/EtherCAT1/=+-EK1100_03_00/=+-ES1004_03_01
//     PlcTask Inputs/GVL_Devices.fb_AT1K0_GAS_PTM_10.i_xAtSpd <-> Channel 2/fb_AT1K0_GAS_PTM_10.i_xAtSpd
//     PlcTask Inputs/GVL_Devices.fb_AT1K0_GAS_PTM_10.i_xDecel <-> Channel 1/fb_AT1K0_GAS_PTM_10.i_xDecel
//     PlcTask Inputs/GVL_Devices.fb_AT1K0_GAS_PTM_10.i_xNCFault <-> Channel 3/fb_AT1K0_GAS_PTM_10.i_xNCFault
//     PlcTask Inputs/GVL_Devices.fb_AT1K0_GAS_PTM_10.i_xRotate <-> Channel 4/fb_AT1K0_GAS_PTM_10.i_xRotate
//   plc_kfe_gatt Instance <-> =+-CX2020/EtherCAT1/=+-EK1100_03_00/=+-ES1004_03_02
//     PlcTask Inputs/GVL_Devices.fb_AT1K0_GAS_PTM_10.i_xAccel <-> Channel 1/fb_AT1K0_GAS_PTM_10.i_xAccel
//   plc_kfe_gatt Instance <-> =+-CX2020/EtherCAT1/=+-EK1100_03_00/=+-ES1004_03_08
//     PlcTask Inputs/GVL_Devices.fb_AT1K0_GAS_PTM_20.i_xAtSpd <-> Channel 2/fb_AT1K0_GAS_PTM_20.i_xAtSpd
//     PlcTask Inputs/GVL_Devices.fb_AT1K0_GAS_PTM_20.i_xDecel <-> Channel 1/fb_AT1K0_GAS_PTM_20.i_xDecel
//     PlcTask Inputs/GVL_Devices.fb_AT1K0_GAS_PTM_20.i_xNCFault <-> Channel 3/fb_AT1K0_GAS_PTM_20.i_xNCFault
//     PlcTask Inputs/GVL_Devices.fb_AT1K0_GAS_PTM_20.i_xRotate <-> Channel 4/fb_AT1K0_GAS_PTM_20.i_xRotate
//   plc_kfe_gatt Instance <-> =+-CX2020/EtherCAT1/=+-EK1100_03_00/=+-ES1004_03_09
//     PlcTask Inputs/GVL_Devices.fb_AT1K0_GAS_PTM_20.i_xAccel <-> Channel 1/fb_AT1K0_GAS_PTM_20.i_xAccel
//   plc_kfe_gatt Instance <-> =+-CX2020/EtherCAT1/=+-EK1100_03_00/=+-ES1004_03_11
//     PlcTask Inputs/GVL_Devices.fb_AT1K0_GAS_PTM_30.i_xAtSpd <-> Channel 2/fb_AT1K0_GAS_PTM_30.i_xAtSpd
//     PlcTask Inputs/GVL_Devices.fb_AT1K0_GAS_PTM_30.i_xDecel <-> Channel 1/fb_AT1K0_GAS_PTM_30.i_xDecel
//     PlcTask Inputs/GVL_Devices.fb_AT1K0_GAS_PTM_30.i_xNCFault <-> Channel 3/fb_AT1K0_GAS_PTM_30.i_xNCFault
//     PlcTask Inputs/GVL_Devices.fb_AT1K0_GAS_PTM_30.i_xRotate <-> Channel 4/fb_AT1K0_GAS_PTM_30.i_xRotate
//   plc_kfe_gatt Instance <-> =+-CX2020/EtherCAT1/=+-EK1100_03_00/=+-ES1004_03_12
//     PlcTask Inputs/GVL_Devices.fb_AT1K0_GAS_PTM_30.i_xAccel <-> Channel 1/fb_AT1K0_GAS_PTM_30.i_xAccel
//   plc_kfe_gatt Instance <-> =+-CX2020/EtherCAT1/=+-EK1100_03_00/=+-ES1004_03_18
//     PlcTask Inputs/GVL_Devices.fb_AT1K0_GAS_PTM_40.i_xAtSpd <-> Channel 2/fb_AT1K0_GAS_PTM_40.i_xAtSpd
//     PlcTask Inputs/GVL_Devices.fb_AT1K0_GAS_PTM_40.i_xDecel <-> Channel 1/fb_AT1K0_GAS_PTM_40.i_xDecel
//     PlcTask Inputs/GVL_Devices.fb_AT1K0_GAS_PTM_40.i_xNCFault <-> Channel 3/fb_AT1K0_GAS_PTM_40.i_xNCFault
//     PlcTask Inputs/GVL_Devices.fb_AT1K0_GAS_PTM_40.i_xRotate <-> Channel 4/fb_AT1K0_GAS_PTM_40.i_xRotate
//   plc_kfe_gatt Instance <-> =+-CX2020/EtherCAT1/=+-EK1100_03_00/=+-ES1004_03_19
//     PlcTask Inputs/GVL_Devices.fb_AT1K0_GAS_PTM_40.i_xAccel <-> Channel 1/fb_AT1K0_GAS_PTM_40.i_xAccel
//   plc_kfe_gatt Instance <-> =+-CX2020/EtherCAT1/=+-EK1100_03_00/=+-ES1004_03_21
//     PlcTask Inputs/GVL_Devices.fb_AT1K0_GAS_VRC_11.i_xClsLS <-> Channel 2/Input
//     PlcTask Inputs/GVL_Devices.fb_AT1K0_GAS_VRC_11.i_xOpnLS <-> Channel 1/Input
//   plc_kfe_gatt Instance <-> =+-CX2020/EtherCAT1/=+-EK1100_03_00/=+-ES3064_03_04
//     PlcTask Inputs/GVL_Devices.fb_AT1K0_GAS_PTM_10.i_iCurrentMon <-> AI Standard Channel 2/fb_AT1K0_GAS_PTM_10.i_iCurrentMon
//     PlcTask Inputs/GVL_Devices.fb_AT1K0_GAS_PTM_10.i_iRawSpeed <-> AI Standard Channel 1/fb_AT1K0_GAS_PTM_10.i_iRawSpeed
//     PlcTask Inputs/GVL_Devices.fb_AT1K0_GAS_PTM_10.i_iTempMon <-> AI Standard Channel 3/fb_AT1K0_GAS_PTM_10.i_iTempMon
//   plc_kfe_gatt Instance <-> =+-CX2020/EtherCAT1/=+-EK1100_03_00/=+-ES3064_03_06
//     PlcTask Inputs/GVL_Devices.fb_AT1K0_GAS_PTM_20.i_iCurrentMon <-> AI Standard Channel 2/fb_AT1K0_GAS_PTM_20.i_iCurrentMon
//     PlcTask Inputs/GVL_Devices.fb_AT1K0_GAS_PTM_20.i_iRawSpeed <-> AI Standard Channel 1/fb_AT1K0_GAS_PTM_20.i_iRawSpeed
//     PlcTask Inputs/GVL_Devices.fb_AT1K0_GAS_PTM_20.i_iTempMon <-> AI Standard Channel 3/fb_AT1K0_GAS_PTM_20.i_iTempMon
//   plc_kfe_gatt Instance <-> =+-CX2020/EtherCAT1/=+-EK1100_03_00/=+-ES3064_03_14
//     PlcTask Inputs/GVL_Devices.fb_AT1K0_GAS_PTM_30.i_iCurrentMon <-> AI Standard Channel 2/fb_AT1K0_GAS_PTM_30.i_iCurrentMon
//     PlcTask Inputs/GVL_Devices.fb_AT1K0_GAS_PTM_30.i_iRawSpeed <-> AI Standard Channel 1/fb_AT1K0_GAS_PTM_30.i_iRawSpeed
//     PlcTask Inputs/GVL_Devices.fb_AT1K0_GAS_PTM_30.i_iTempMon <-> AI Standard Channel 3/fb_AT1K0_GAS_PTM_30.i_iTempMon
//   plc_kfe_gatt Instance <-> =+-CX2020/EtherCAT1/=+-EK1100_03_00/=+-ES3064_03_16
//     PlcTask Inputs/GVL_Devices.fb_AT1K0_GAS_PTM_40.i_iCurrentMon <-> AI Standard Channel 2/fb_AT1K0_GAS_PTM_40.i_iCurrentMon
//     PlcTask Inputs/GVL_Devices.fb_AT1K0_GAS_PTM_40.i_iRawSpeed <-> AI Standard Channel 1/fb_AT1K0_GAS_PTM_40.i_iRawSpeed
//     PlcTask Inputs/GVL_Devices.fb_AT1K0_GAS_PTM_40.i_iTempMon <-> AI Standard Channel 3/fb_AT1K0_GAS_PTM_40.i_iTempMon
//   plc_kfe_gatt Instance <-> =+-CX2020/EtherCAT1/=+-EK1100_03_00/=+-ES4004_03_05
//     PlcTask Outputs/GVL_Devices.fb_AT1K0_GAS_PTM_10.q_iSpeedSet <-> AO Outputs Channel 1/fb_AT1K0_GAS_PTM_10.q_iSpeedSet
//     PlcTask Outputs/GVL_Devices.fb_AT1K0_GAS_PTM_20.q_iSpeedSet <-> AO Outputs Channel 3/fb_AT1K0_GAS_PTM_20.q_iSpeedSet
//   plc_kfe_gatt Instance <-> =+-CX2020/EtherCAT1/=+-EK1100_03_00/=+-ES4004_03_15
//     PlcTask Outputs/GVL_Devices.fb_AT1K0_GAS_PTM_30.q_iSpeedSet <-> AO Outputs Channel 1/fb_AT1K0_GAS_PTM_30.q_iSpeedSet
//     PlcTask Outputs/GVL_Devices.fb_AT1K0_GAS_PTM_40.q_iSpeedSet <-> AO Outputs Channel 3/fb_AT1K0_GAS_PTM_40.q_iSpeedSet
//   plc_kfe_gatt Instance <-> =+-CX2020/EtherCAT1/=+-EK1100_04_00/=+-EL2212_04_18
//     PlcTask Inputs/DIAGNOSTICS.DRL_04.SC <-> DOX Synchron info data Channel 2/Info data 1
//     PlcTask Inputs/DIAGNOSTICS.DRL_04.SV <-> DOX Synchron info data Channel 1/Info data 2
//     PlcTask Inputs/DIAGNOSTICS.DRL_04.TEMP <-> DOX Synchron info data Channel 1/Info data 1
//     PlcTask Outputs/GVL_Devices.fb_AT1K0_GAS_VVC_80.q_xOPN_DO <-> DOX Control Channel 2/Control/Output
//   plc_kfe_gatt Instance <-> =+-CX2020/EtherCAT1/=+-EK1100_04_00/=+-EL3174_04_17
//     PlcTask Inputs/GVL_Devices.GCM_70.i_iPRESS_R <-> AI Standard Channel 3/GCM_70.i_iPRESS_R
//     PlcTask Inputs/GVL_Devices.GCM_80.i_iPRESS_R <-> AI Standard Channel 1/GCM_80.i_iPRESS_R
//     PlcTask Inputs/GVL_Devices.GCM_81.i_iPRESS_R <-> AI Standard Channel 2/Value
//   plc_kfe_gatt Instance <-> =+-CX2020/EtherCAT1/=+-EK1100_04_00/=+-EL7041_04_07
//     PlcTask Inputs/Main.M5.bLimitBackwardEnable <-> STM Status/Status/Digital input 1
//     PlcTask Inputs/Main.M5.bLimitForwardEnable <-> STM Status/Status/Digital input 2
//   plc_kfe_gatt Instance <-> =+-CX2020/EtherCAT1/=+-EK1100_04_00/=+-EL7041_04_08
//     PlcTask Inputs/Main.M6.bLimitBackwardEnable <-> STM Status/Status/Digital input 1
//     PlcTask Inputs/Main.M6.bLimitForwardEnable <-> STM Status/Status/Digital input 2
//   plc_kfe_gatt Instance <-> =+-CX2020/EtherCAT1/=+-EK1100_04_00/=+-EL7041_04_10
//     PlcTask Inputs/Main.M7.bLimitBackwardEnable <-> STM Status/Status/Digital input 1
//     PlcTask Inputs/Main.M7.bLimitForwardEnable <-> STM Status/Status/Digital input 2
//   plc_kfe_gatt Instance <-> =+-CX2020/EtherCAT1/=+-EK1100_04_00/=+-EL7041_04_11
//     PlcTask Inputs/Main.M8.bLimitBackwardEnable <-> STM Status/Status/Digital input 1
//     PlcTask Inputs/Main.M8.bLimitForwardEnable <-> STM Status/Status/Digital input 2
//   plc_kfe_gatt Instance <-> =+-CX2020/EtherCAT1/=+-EK1100_04_00/=+-ES1084_04_06
//     PlcTask Inputs/GVL_Devices.fb_AT1K0_GAS_PTM_80.i_xAtSpd <-> Channel 1/fb_AT1K0_GAS_PTM_80.i_xAtSpd
//     PlcTask Inputs/GVL_Devices.fb_AT1K0_GAS_PTM_80.i_xFault <-> Channel 2/fb_AT1K0_GAS_PTM_80.i_xFault
//   plc_kfe_gatt Instance <-> =+-CX2020/EtherCAT1/=+-EK1100_04_00/=+-ES2004_04_01
//     PlcTask Outputs/GVL_Devices.VVC_71.q_xOPN_DO <-> Channel 1/VVC_71.q_xOPN_DO
//     PlcTask Outputs/GVL_Devices.VVC_72.q_xOPN_DO <-> Channel 2/VVC_72.q_xOPN_DO
//     PlcTask Outputs/GVL_Devices.fb_AT1K0_GAS_PTM_80.q_RunDO <-> Channel 3/fb_AT1K0_GAS_PTM_80.q_RunDO
//   plc_kfe_gatt Instance <-> =+-CX2020/EtherCAT1/=+-EK1100_04_00/=+-ES2004_04_09
//     PlcTask Outputs/Main.M{5..8}.bBrakeRelease <-> Channel {1..4}/Output  (4 links)
//   plc_kfe_gatt Instance <-> =+-CX2020/EtherCAT1/=+-EK1100_04_00/=+-ES4004_04_02
//     PlcTask Outputs/GVL_Devices.VCN_70.q_iRawPosition <-> AO Outputs Channel 1/VCN_70.q_iRawPosition
//   plc_kfe_gatt Instance <-> =+-CX2020/EtherCAT1/=+-EK1100_05_00/=+-EL1084_05_12
//     PlcTask Inputs/GVL_Devices.fb_AT1K0_GAS_PMF_110.i_xAlarmOK <-> Channel 2/fb_AT1K0_GAS_PMF_110.i_xAlarmOK
//     PlcTask Inputs/GVL_Devices.fb_AT1K0_GAS_PMF_120.i_xAlarmOK <-> Channel 4/fb_AT1K0_GAS_PMF_120.i_xAlarmOK
//     PlcTask Inputs/GVL_Devices.fb_AT1K0_GAS_PMF_110.i_xIsRun <-> Channel 1/fb_AT1K0_GAS_PMF_110.i_xIsRun
//     PlcTask Inputs/GVL_Devices.fb_AT1K0_GAS_PMF_120.i_xIsRun <-> Channel 3/fb_AT1K0_GAS_PMF_120.i_xIsRun
//   plc_kfe_gatt Instance <-> =+-CX2020/EtherCAT1/=+-EK1100_05_00/=+-EL1084_05_13
//     PlcTask Inputs/GVL_Devices.fb_AT1K0_GAS_PMF_140.i_xAlarmOK <-> Channel 2/fb_AT1K0_GAS_PMF_140.i_xAlarmOK
//     PlcTask Inputs/GVL_Devices.fb_AT1K0_GAS_PMF_140.i_xIsRun <-> Channel 1/fb_AT1K0_GAS_PMF_140.i_xIsRun
//   plc_kfe_gatt Instance <-> =+-CX2020/EtherCAT1/=+-EK1100_05_00/=+-EL2212_05_09
//     PlcTask Inputs/DIAGNOSTICS.DRL_05.SC <-> DOX Synchron info data Channel 2/Info data 1
//     PlcTask Inputs/DIAGNOSTICS.DRL_05.SV <-> DOX Synchron info data Channel 1/Info data 2
//     PlcTask Inputs/DIAGNOSTICS.DRL_05.TEMP <-> DOX Synchron info data Channel 1/Info data 1
//   plc_kfe_gatt Instance <-> =+-CX2020/EtherCAT1/=+-EK1100_05_00/=+-EL2798_05_10
//     PlcTask Outputs/GVL_Devices.fb_AT1K0_GAS_PMF_110.q_xResetAlarm <-> Channel 2/fb_AT1K0_GAS_PMF_110.q_xResetAlarm
//     PlcTask Outputs/GVL_Devices.fb_AT1K0_GAS_PMF_120.q_xResetAlarm <-> Channel 4/fb_AT1K0_GAS_PMF_120.q_xResetAlarm
//     PlcTask Outputs/GVL_Devices.fb_AT1K0_GAS_PMF_140.q_xResetAlarm <-> Channel 6/fb_AT1K0_GAS_PMF_140.q_xResetAlarm
//     PlcTask Outputs/GVL_Devices.fb_AT1K0_GAS_PMF_110.q_xRunDo <-> Channel 1/fb_AT1K0_GAS_PMF_110.q_xRunDo
//     PlcTask Outputs/GVL_Devices.fb_AT1K0_GAS_PMF_120.q_xRunDo <-> Channel 3/fb_AT1K0_GAS_PMF_120.q_xRunDo
//     PlcTask Outputs/GVL_Devices.fb_AT1K0_GAS_PMF_140.q_xRunDo <-> Channel 5/fb_AT1K0_GAS_PMF_140.q_xRunDo
//   plc_kfe_gatt Instance <-> =+-CX2020/EtherCAT1/=+-EK1100_05_00/=+-EL3174_05_16
//     PlcTask Inputs/GVL_Devices.fb_AT1K0_GAS_GPI_111.i_iPRESS_R <-> AI Standard Channel 1/fb_AT1K0_GAS_GPI_111.i_iPRESS_R
//     PlcTask Inputs/GVL_Devices.fb_AT1K0_GAS_GPI_141.i_iPRESS_R <-> AI Standard Channel 3/fb_AT1K0_GAS_GPI_141.i_iPRESS_R
//     PlcTask Inputs/GVL_Devices.fb_AT1K0_GAS_GPI_121.i_iPRESS_R <-> AI Standard Channel 2/Value
//   plc_kfe_gatt Instance <-> =+-CX2020/EtherCAT1/=+-EK1100_05_00/=+-ES1004_05_01
//     PlcTask Inputs/GVL_Devices.fb_AT1K0_GAS_VRC_70.i_xClsLS <-> Channel 2/fb_AT1K0_GAS_VRC_70.i_xClsLS
//     PlcTask Inputs/GVL_Devices.fb_AT1K0_GAS_VRC_80.i_xClsLS <-> Channel 4/fb_AT1K0_GAS_VRC_80.i_xClsLS
//     PlcTask Inputs/GVL_Devices.fb_AT1K0_GAS_VRC_70.i_xOpnLS <-> Channel 1/fb_AT1K0_GAS_VRC_70.i_xOpnLS
//     PlcTask Inputs/GVL_Devices.fb_AT1K0_GAS_VRC_80.i_xOpnLS <-> Channel 3/fb_AT1K0_GAS_VRC_80.i_xOpnLS
//   plc_kfe_gatt Instance <-> =+-CX2020/EtherCAT1/=+-EK1100_05_00/=+-ES1004_05_03
//     PlcTask Inputs/GVL_Devices.fb_AT1K0_GAS_VRC_100.i_xClsLS <-> Channel 4/fb_AT1K0_GAS_VRC_100.i_xClsLS
//     PlcTask Inputs/GVL_Devices.fb_AT1K0_GAS_VRC_90.i_xClsLS <-> Channel 2/fb_AT1K0_GAS_VRC_90.i_xClsLS
//     PlcTask Inputs/GVL_Devices.fb_AT1K0_GAS_VRC_100.i_xOpnLS <-> Channel 3/fb_AT1K0_GAS_VRC_100.i_xOpnLS
//     PlcTask Inputs/GVL_Devices.fb_AT1K0_GAS_VRC_90.i_xOpnLS <-> Channel 1/fb_AT1K0_GAS_VRC_90.i_xOpnLS
//   plc_kfe_gatt Instance <-> =+-CX2020/EtherCAT1/=+-EK1100_05_00/=+-ES1004_05_06
//     PlcTask Inputs/GVL_Devices.fb_AT1K0_GAS_VRC_110.i_xClsLS <-> Channel 2/fb_AT1K0_GAS_VRC_110.i_xClsLS
//     PlcTask Inputs/GVL_Devices.fb_AT1K0_GAS_VRC_120.i_xClsLS <-> Channel 4/fb_AT1K0_GAS_VRC_120.i_xClsLS
//     PlcTask Inputs/GVL_Devices.fb_AT1K0_GAS_VRC_110.i_xOpnLS <-> Channel 1/fb_AT1K0_GAS_VRC_110.i_xOpnLS
//     PlcTask Inputs/GVL_Devices.fb_AT1K0_GAS_VRC_120.i_xOpnLS <-> Channel 3/fb_AT1K0_GAS_VRC_120.i_xOpnLS
//   plc_kfe_gatt Instance <-> =+-CX2020/EtherCAT1/=+-EK1100_05_00/=+-ES1004_05_08
//     PlcTask Inputs/GVL_Devices.fb_AT1K0_GAS_VRC_130.i_xClsLS <-> Channel 2/fb_AT1K0_GAS_VRC_130.i_xClsLS
//     PlcTask Inputs/GVL_Devices.fb_AT1K0_GAS_VRC_140.i_xClsLS <-> Channel 4/fb_AT1K0_GAS_VRC_140.i_xClsLS
//     PlcTask Inputs/GVL_Devices.fb_AT1K0_GAS_VRC_130.i_xOpnLS <-> Channel 1/fb_AT1K0_GAS_VRC_130.i_xOpnLS
//     PlcTask Inputs/GVL_Devices.fb_AT1K0_GAS_VRC_140.i_xOpnLS <-> Channel 3/fb_AT1K0_GAS_VRC_140.i_xOpnLS
//   plc_kfe_gatt Instance <-> =+-CX2020/EtherCAT1/=+-EK1100_05_00/=+-ES2004_05_02
//     PlcTask Outputs/GVL_Devices.fb_AT1K0_GAS_VRC_70.q_xOPN_DO <-> Channel 1/fb_AT1K0_GAS_VRC_70.q_xOPN_DO
//     PlcTask Outputs/GVL_Devices.fb_AT1K0_GAS_VRC_80.q_xOPN_DO <-> Channel 2/fb_AT1K0_GAS_VRC_80.q_xOPN_DO
//     PlcTask Outputs/GVL_Devices.fb_AT1K0_GAS_VVC_110.q_xOPN_DO <-> Channel 3/Output
//     PlcTask Outputs/GVL_Devices.fb_AT1K0_GAS_VVC_120.q_xOPN_DO <-> Channel 4/Output
//   plc_kfe_gatt Instance <-> =+-CX2020/EtherCAT1/=+-EK1100_05_00/=+-ES2004_05_04
//     PlcTask Outputs/GVL_Devices.fb_AT1K0_GAS_VRC_100.q_xOPN_DO <-> Channel 2/fb_AT1K0_GAS_VRC_100.q_xOPN_DO
//     PlcTask Outputs/GVL_Devices.fb_AT1K0_GAS_VRC_90.q_xOPN_DO <-> Channel 1/fb_AT1K0_GAS_VRC_90.q_xOPN_DO
//     PlcTask Outputs/GVL_Devices.fb_AT1K0_GAS_VVC_140.q_xOPN_DO <-> Channel 3/Output
//   plc_kfe_gatt Instance <-> =+-CX2020/EtherCAT1/=+-EK1100_05_00/=+-ES2004_05_05
//     PlcTask Outputs/GVL_Devices.fb_AT1K0_GAS_VRC_110.q_xOPN_DO <-> Channel 1/fb_AT1K0_GAS_VRC_110.q_xOPN_DO
//     PlcTask Outputs/GVL_Devices.fb_AT1K0_GAS_VRC_120.q_xOPN_DO <-> Channel 2/fb_AT1K0_GAS_VRC_120.q_xOPN_DO
//   plc_kfe_gatt Instance <-> =+-CX2020/EtherCAT1/=+-EK1100_05_00/=+-ES2004_05_07
//     PlcTask Outputs/GVL_Devices.fb_AT1K0_GAS_VRC_130.q_xOPN_DO <-> Channel 1/fb_AT1K0_GAS_VRC_130.q_xOPN_DO
//     PlcTask Outputs/GVL_Devices.fb_AT1K0_GAS_VRC_140.q_xOPN_DO <-> Channel 2/fb_AT1K0_GAS_VRC_140.q_xOPN_DO
//   plc_kfe_gatt Instance <-> =+-CX2020/EtherCAT1/=+-EK1100_06_00/=+-EL2212_06_25
//     PlcTask Inputs/DIAGNOSTICS.DRL_06.SC <-> DOX Synchron info data Channel 2/Info data 1
//     PlcTask Inputs/DIAGNOSTICS.DRL_06.SV <-> DOX Synchron info data Channel 1/Info data 2
//     PlcTask Inputs/DIAGNOSTICS.DRL_06.TEMP <-> DOX Synchron info data Channel 1/Info data 1
//   plc_kfe_gatt Instance <-> =+-CX2020/EtherCAT1/=+-EK1100_06_00/=+-EL2794_06_22
//     PlcTask Outputs/GVL_Devices.fb_AT1K0_GAS_PMF_100.q_xBPStart <-> Channel 4/fb_AT1K0_GAS_PMF_100.q_xBPStart
//     PlcTask Outputs/GVL_Devices.fb_AT1K0_GAS_PMF_90.q_xBPStart <-> Channel 2/fb_AT1K0_GAS_PMF_90.q_xBPStart
//     PlcTask Outputs/GVL_Devices.fb_AT1K0_GAS_PMF_100.q_xMPStart <-> Channel 3/fb_AT1K0_GAS_PMF_100.q_xMPStart
//     PlcTask Outputs/GVL_Devices.fb_AT1K0_GAS_PMF_90.q_xMPStart <-> Channel 1/fb_AT1K0_GAS_PMF_90.q_xMPStart
//   plc_kfe_gatt Instance <-> =+-CX2020/EtherCAT1/=+-EK1100_06_00/=+-EL2798_06_03
//     PlcTask Outputs/GVL_Devices.fb_AT1K0_GAS_PTM_110.q_xProtection <-> Channel 5/fb_AT1K0_GAS_PTM_110.q_xProtection
//     PlcTask Outputs/GVL_Devices.fb_AT1K0_GAS_PTM_110.q_xReset <-> Channel 1/fb_AT1K0_GAS_PTM_110.q_xReset
//     PlcTask Outputs/GVL_Devices.fb_AT1K0_GAS_PTM_110.q_xSetSpeed <-> Channel 4/fb_AT1K0_GAS_PTM_110.q_xSetSpeed
//     PlcTask Outputs/GVL_Devices.fb_AT1K0_GAS_PTM_110.q_xStart <-> Channel 2/fb_AT1K0_GAS_PTM_110.q_xStart
//     PlcTask Outputs/GVL_Devices.fb_AT1K0_GAS_PTM_110.q_xStop <-> Channel 3/fb_AT1K0_GAS_PTM_110.q_xStop
//   plc_kfe_gatt Instance <-> =+-CX2020/EtherCAT1/=+-EK1100_06_00/=+-EL2798_06_07
//     PlcTask Outputs/GVL_Devices.fb_AT1K0_GAS_PTM_120.q_xProtection <-> Channel 4/fb_AT1K0_GAS_PTM_120.q_xProtection
//     PlcTask Outputs/GVL_Devices.fb_AT1K0_GAS_PTM_120.q_xReset <-> Channel 1/fb_AT1K0_GAS_PTM_120.q_xReset
//     PlcTask Outputs/GVL_Devices.fb_AT1K0_GAS_PTM_120.q_xSetSpeed <-> Channel 5/fb_AT1K0_GAS_PTM_120.q_xSetSpeed
//     PlcTask Outputs/GVL_Devices.fb_AT1K0_GAS_PTM_120.q_xStart <-> Channel 2/fb_AT1K0_GAS_PTM_120.q_xStart
//     PlcTask Outputs/GVL_Devices.fb_AT1K0_GAS_PTM_120.q_xStop <-> Channel 3/fb_AT1K0_GAS_PTM_120.q_xStop
//   plc_kfe_gatt Instance <-> =+-CX2020/EtherCAT1/=+-EK1100_06_00/=+-EL2798_06_13
//     PlcTask Outputs/GVL_Devices.fb_AT1K0_GAS_PTM_130.q_xProtection <-> Channel 4/fb_AT1K0_GAS_PTM_130.q_xProtection
//     PlcTask Outputs/GVL_Devices.fb_AT1K0_GAS_PTM_130.q_xReset <-> Channel 1/fb_AT1K0_GAS_PTM_130.q_xReset
//     PlcTask Outputs/GVL_Devices.fb_AT1K0_GAS_PTM_130.q_xSetSpeed <-> Channel 5/fb_AT1K0_GAS_PTM_130.q_xSetSpeed
//     PlcTask Outputs/GVL_Devices.fb_AT1K0_GAS_PTM_130.q_xStart <-> Channel 2/fb_AT1K0_GAS_PTM_130.q_xStart
//     PlcTask Outputs/GVL_Devices.fb_AT1K0_GAS_PTM_130.q_xStop <-> Channel 3/fb_AT1K0_GAS_PTM_130.q_xStop
//   plc_kfe_gatt Instance <-> =+-CX2020/EtherCAT1/=+-EK1100_06_00/=+-EL2798_06_17
//     PlcTask Outputs/GVL_Devices.fb_AT1K0_GAS_PTM_140.q_xProtection <-> Channel 4/fb_AT1K0_GAS_PTM_140.q_xProtection
//     PlcTask Outputs/GVL_Devices.fb_AT1K0_GAS_PTM_140.q_xReset <-> Channel 1/fb_AT1K0_GAS_PTM_140.q_xReset
//     PlcTask Outputs/GVL_Devices.fb_AT1K0_GAS_PTM_140.q_xSetSpeed <-> Channel 5/fb_AT1K0_GAS_PTM_140.q_xSetSpeed
//     PlcTask Outputs/GVL_Devices.fb_AT1K0_GAS_PTM_140.q_xStart <-> Channel 2/fb_AT1K0_GAS_PTM_140.q_xStart
//     PlcTask Outputs/GVL_Devices.fb_AT1K0_GAS_PTM_140.q_xStop <-> Channel 3/fb_AT1K0_GAS_PTM_140.q_xStop
//   plc_kfe_gatt Instance <-> =+-CX2020/EtherCAT1/=+-EK1100_06_00/=+-ES1004_06_01
//     PlcTask Inputs/GVL_Devices.fb_AT1K0_GAS_PTM_110.i_xAccel <-> Channel 4/fb_AT1K0_GAS_PTM_110.i_xAccel
//     PlcTask Inputs/GVL_Devices.fb_AT1K0_GAS_PTM_110.i_xAtSpd <-> Channel 1/fb_AT1K0_GAS_PTM_110.i_xAtSpd
//     PlcTask Inputs/GVL_Devices.fb_AT1K0_GAS_PTM_110.i_xFaultNC <-> Channel 2/fb_AT1K0_GAS_PTM_110.i_xFaultNC
//     PlcTask Inputs/GVL_Devices.fb_AT1K0_GAS_PTM_110.i_xRotate <-> Channel 3/fb_AT1K0_GAS_PTM_110.i_xRotate
//   plc_kfe_gatt Instance <-> =+-CX2020/EtherCAT1/=+-EK1100_06_00/=+-ES1004_06_02
//     PlcTask Inputs/GVL_Devices.fb_AT1K0_GAS_PTM_110.i_xDecel <-> Channel 1/fb_AT1K0_GAS_PTM_110.i_xDecel
//   plc_kfe_gatt Instance <-> =+-CX2020/EtherCAT1/=+-EK1100_06_00/=+-ES1004_06_08
//     PlcTask Inputs/GVL_Devices.fb_AT1K0_GAS_PTM_120.i_xAtSpd <-> Channel 2/fb_AT1K0_GAS_PTM_120.i_xAtSpd
//     PlcTask Inputs/GVL_Devices.fb_AT1K0_GAS_PTM_120.i_xDecel <-> Channel 1/fb_AT1K0_GAS_PTM_120.i_xDecel
//     PlcTask Inputs/GVL_Devices.fb_AT1K0_GAS_PTM_120.i_xNCFault <-> Channel 3/fb_AT1K0_GAS_PTM_120.i_xNCFault
//     PlcTask Inputs/GVL_Devices.fb_AT1K0_GAS_PTM_120.i_xRotate <-> Channel 4/fb_AT1K0_GAS_PTM_120.i_xRotate
//   plc_kfe_gatt Instance <-> =+-CX2020/EtherCAT1/=+-EK1100_06_00/=+-ES1004_06_09
//     PlcTask Inputs/GVL_Devices.fb_AT1K0_GAS_PTM_120.i_xAccel <-> Channel 1/fb_AT1K0_GAS_PTM_120.i_xAccel
//   plc_kfe_gatt Instance <-> =+-CX2020/EtherCAT1/=+-EK1100_06_00/=+-ES1004_06_11
//     PlcTask Inputs/GVL_Devices.fb_AT1K0_GAS_PTM_130.i_xAtSpd <-> Channel 2/fb_AT1K0_GAS_PTM_130.i_xAtSpd
//     PlcTask Inputs/GVL_Devices.fb_AT1K0_GAS_PTM_130.i_xDecel <-> Channel 1/fb_AT1K0_GAS_PTM_130.i_xDecel
//     PlcTask Inputs/GVL_Devices.fb_AT1K0_GAS_PTM_130.i_xNCFault <-> Channel 3/fb_AT1K0_GAS_PTM_130.i_xNCFault
//     PlcTask Inputs/GVL_Devices.fb_AT1K0_GAS_PTM_130.i_xRotate <-> Channel 4/fb_AT1K0_GAS_PTM_130.i_xRotate
//   plc_kfe_gatt Instance <-> =+-CX2020/EtherCAT1/=+-EK1100_06_00/=+-ES1004_06_12
//     PlcTask Inputs/GVL_Devices.fb_AT1K0_GAS_PTM_130.i_xAccel <-> Channel 1/fb_AT1K0_GAS_PTM_130.i_xAccel
//   plc_kfe_gatt Instance <-> =+-CX2020/EtherCAT1/=+-EK1100_06_00/=+-ES1004_06_18
//     PlcTask Inputs/GVL_Devices.fb_AT1K0_GAS_PTM_140.i_xAtSpd <-> Channel 2/fb_AT1K0_GAS_PTM_140.i_xAtSpd
//     PlcTask Inputs/GVL_Devices.fb_AT1K0_GAS_PTM_140.i_xDecel <-> Channel 1/fb_AT1K0_GAS_PTM_140.i_xDecel
//     PlcTask Inputs/GVL_Devices.fb_AT1K0_GAS_PTM_140.i_xNCFault <-> Channel 3/fb_AT1K0_GAS_PTM_140.i_xNCFault
//     PlcTask Inputs/GVL_Devices.fb_AT1K0_GAS_PTM_140.i_xRotate <-> Channel 4/fb_AT1K0_GAS_PTM_140.i_xRotate
//   plc_kfe_gatt Instance <-> =+-CX2020/EtherCAT1/=+-EK1100_06_00/=+-ES1004_06_19
//     PlcTask Inputs/GVL_Devices.fb_AT1K0_GAS_PTM_140.i_xAccel <-> Channel 1/fb_AT1K0_GAS_PTM_140.i_xAccel
//   plc_kfe_gatt Instance <-> =+-CX2020/EtherCAT1/=+-EK1100_06_00/=+-ES1088_06_20
//     PlcTask Inputs/GVL_Devices.fb_AT1K0_GAS_PMF_90.i_xAlarmOK <-> Channel 4/fb_AT1K0_GAS_PMF_90.i_xAlarmOK
//     PlcTask Inputs/GVL_Devices.fb_AT1K0_GAS_PMF_90.i_xBPStatus <-> Channel 2/fb_AT1K0_GAS_PMF_90.i_xBPStatus
//     PlcTask Inputs/GVL_Devices.fb_AT1K0_GAS_PMF_90.i_xMPStatus <-> Channel 1/fb_AT1K0_GAS_PMF_90.i_xMPStatus
//     PlcTask Inputs/GVL_Devices.fb_AT1K0_GAS_PMF_90.i_xRemote <-> Channel 5/fb_AT1K0_GAS_PMF_90.i_xRemote
//     PlcTask Inputs/GVL_Devices.fb_AT1K0_GAS_PMF_90.i_xWarning <-> Channel 3/fb_AT1K0_GAS_PMF_90.i_xWarning
//   plc_kfe_gatt Instance <-> =+-CX2020/EtherCAT1/=+-EK1100_06_00/=+-ES1088_06_23
//     PlcTask Inputs/GVL_Devices.fb_AT1K0_GAS_PMF_100.i_xAlarmOK <-> Channel 4/fb_AT1K0_GAS_PMF_100.i_xAlarmOK
//     PlcTask Inputs/GVL_Devices.fb_AT1K0_GAS_PMF_100.i_xBPStatus <-> Channel 2/fb_AT1K0_GAS_PMF_100.i_xBPStatus
//     PlcTask Inputs/GVL_Devices.fb_AT1K0_GAS_PMF_100.i_xMPStatus <-> Channel 1/fb_AT1K0_GAS_PMF_100.i_xMPStatus
//     PlcTask Inputs/GVL_Devices.fb_AT1K0_GAS_PMF_100.i_xRemote <-> Channel 5/fb_AT1K0_GAS_PMF_100.i_xRemote
//     PlcTask Inputs/GVL_Devices.fb_AT1K0_GAS_PMF_100.i_xWarning <-> Channel 3/fb_AT1K0_GAS_PMF_100.i_xWarning
//   plc_kfe_gatt Instance <-> =+-CX2020/EtherCAT1/=+-EK1100_06_00/=+-ES3064_06_04
//     PlcTask Inputs/GVL_Devices.fb_AT1K0_GAS_PTM_110.i_iRawSpeed <-> AI Standard Channel 1/fb_AT1K0_GAS_PTM_110.i_iRawSpeed
//   plc_kfe_gatt Instance <-> =+-CX2020/EtherCAT1/=+-EK1100_06_00/=+-ES3064_06_06
//     PlcTask Inputs/GVL_Devices.fb_AT1K0_GAS_PTM_120.i_iCurrentMon <-> AI Standard Channel 2/fb_AT1K0_GAS_PTM_120.i_iCurrentMon
//     PlcTask Inputs/GVL_Devices.fb_AT1K0_GAS_PTM_120.i_iRawSpeed <-> AI Standard Channel 1/fb_AT1K0_GAS_PTM_120.i_iRawSpeed
//     PlcTask Inputs/GVL_Devices.fb_AT1K0_GAS_PTM_120.i_iTempMon <-> AI Standard Channel 3/fb_AT1K0_GAS_PTM_120.i_iTempMon
//   plc_kfe_gatt Instance <-> =+-CX2020/EtherCAT1/=+-EK1100_06_00/=+-ES3064_06_14
//     PlcTask Inputs/GVL_Devices.fb_AT1K0_GAS_PTM_130.i_iCurrentMon <-> AI Standard Channel 2/fb_AT1K0_GAS_PTM_130.i_iCurrentMon
//     PlcTask Inputs/GVL_Devices.fb_AT1K0_GAS_PTM_130.i_iRawSpeed <-> AI Standard Channel 1/fb_AT1K0_GAS_PTM_130.i_iRawSpeed
//     PlcTask Inputs/GVL_Devices.fb_AT1K0_GAS_PTM_130.i_iTempMon <-> AI Standard Channel 3/fb_AT1K0_GAS_PTM_130.i_iTempMon
//   plc_kfe_gatt Instance <-> =+-CX2020/EtherCAT1/=+-EK1100_06_00/=+-ES3064_06_16
//     PlcTask Inputs/GVL_Devices.fb_AT1K0_GAS_PTM_140.i_iCurrentMon <-> AI Standard Channel 2/fb_AT1K0_GAS_PTM_140.i_iCurrentMon
//     PlcTask Inputs/GVL_Devices.fb_AT1K0_GAS_PTM_140.i_iRawSpeed <-> AI Standard Channel 1/fb_AT1K0_GAS_PTM_140.i_iRawSpeed
//     PlcTask Inputs/GVL_Devices.fb_AT1K0_GAS_PTM_140.i_iTempMon <-> AI Standard Channel 3/fb_AT1K0_GAS_PTM_140.i_iTempMon
//   plc_kfe_gatt Instance <-> =+-CX2020/EtherCAT1/=+-EK1100_06_00/=+-ES4004_06_05
//     PlcTask Outputs/GVL_Devices.fb_AT1K0_GAS_PTM_110.q_iSpeedSet <-> AO Outputs Channel 1/fb_AT1K0_GAS_PTM_110.q_iSpeedSet
//     PlcTask Outputs/GVL_Devices.fb_AT1K0_GAS_PTM_120.q_iSpeedSet <-> AO Outputs Channel 3/fb_AT1K0_GAS_PTM_120.q_iSpeedSet
//   plc_kfe_gatt Instance <-> =+-CX2020/EtherCAT1/=+-EK1100_06_00/=+-ES4004_06_15
//     PlcTask Outputs/GVL_Devices.fb_AT1K0_GAS_PTM_130.q_iSpeedSet <-> AO Outputs Channel 1/fb_AT1K0_GAS_PTM_130.q_iSpeedSet
//     PlcTask Outputs/GVL_Devices.fb_AT1K0_GAS_PTM_140.q_iSpeedSet <-> AO Outputs Channel 3/fb_AT1K0_GAS_PTM_140.q_iSpeedSet
//   plc_kfe_gatt Instance <-> =+-CX2020/EtherCAT1/=+-EK1200_00_00/=+-ES2202_00_07
//     PlcTask Outputs/GVL_PMPS.g_FastFaultOutput1.q_xFastFaultOut <-> Channel 1/Output
//     PlcTask Outputs/GVL_PMPS.g_FastFaultOutput2.q_xFastFaultOut <-> Channel 2/Output
//   plc_kfe_gatt Instance <-> =+-CX2020/EtherCAT1/=+-EK1200_00_00/PMPS_PRE
//     PlcTask Inputs/GVL_PMPS.Req_Trans <-> IO Inputs/Requested Transmission
//     PlcTask Inputs/PRG_PMPS.fbArbiterIO.i_stCurrentBP <-> IO Inputs/CurrentBP
//     PlcTask Inputs/PRG_PMPS.fbArbiterIO.xTxPDO_state <-> SYNC Inputs/TxPDO state
//     PlcTask Inputs/PRG_PMPS.fbArbiterIO.xTxPDO_toggle <-> SYNC Inputs/TxPDO toggle
//     PlcTask Outputs/GVL_PMPS.Cur_Trans <-> IO Outputs/Current Transmission
//     PlcTask Outputs/GVL_PMPS.bStatus <-> IO Outputs/bGattStatus
//     PlcTask Outputs/PRG_PMPS.fbArbiterIO.q_stRequestedBP <-> IO Outputs/RequestedBP
//   plc_kfe_gatt Instance <-> NC-Task 1 SAF/Axes/MA_1_X
//     PlcTask Inputs/Main.M1.Axis.NcToPlc <-> Outputs/ToPlc
//     PlcTask Outputs/Main.M1.Axis.PlcToNc <-> Inputs/FromPlc
//   plc_kfe_gatt Instance <-> NC-Task 1 SAF/Axes/MA_1_Y
//     PlcTask Inputs/Main.M2.Axis.NcToPlc <-> Outputs/ToPlc
//     PlcTask Outputs/Main.M2.Axis.PlcToNc <-> Inputs/FromPlc
//   plc_kfe_gatt Instance <-> NC-Task 1 SAF/Axes/MA_2_X
//     PlcTask Inputs/Main.M3.Axis.NcToPlc <-> Outputs/ToPlc
//     PlcTask Outputs/Main.M3.Axis.PlcToNc <-> Inputs/FromPlc
//   plc_kfe_gatt Instance <-> NC-Task 1 SAF/Axes/MA_2_Y
//     PlcTask Inputs/Main.M4.Axis.NcToPlc <-> Outputs/ToPlc
//     PlcTask Outputs/Main.M4.Axis.PlcToNc <-> Inputs/FromPlc
//   plc_kfe_gatt Instance <-> NC-Task 1 SAF/Axes/MA_3_X
//     PlcTask Inputs/Main.M5.Axis.NcToPlc <-> Outputs/ToPlc
//     PlcTask Outputs/Main.M5.Axis.PlcToNc <-> Inputs/FromPlc
//   plc_kfe_gatt Instance <-> NC-Task 1 SAF/Axes/MA_3_Y
//     PlcTask Inputs/Main.M6.Axis.NcToPlc <-> Outputs/ToPlc
//     PlcTask Outputs/Main.M6.Axis.PlcToNc <-> Inputs/FromPlc
//   plc_kfe_gatt Instance <-> NC-Task 1 SAF/Axes/MA_4_X
//     PlcTask Inputs/Main.M7.Axis.NcToPlc <-> Outputs/ToPlc
//     PlcTask Outputs/Main.M7.Axis.PlcToNc <-> Inputs/FromPlc
//   plc_kfe_gatt Instance <-> NC-Task 1 SAF/Axes/MA_4_Y
//     PlcTask Inputs/Main.M8.Axis.NcToPlc <-> Outputs/ToPlc
//     PlcTask Outputs/Main.M8.Axis.PlcToNc <-> Inputs/FromPlc
//   plc_kfe_gatt Instance <-> NC-Task 1 SAF/Axes/VGP_80
//     PlcTask Inputs/GVL_Devices.VGP_80.Axis.NcToPlc <-> Outputs/ToPlc
//     PlcTask Outputs/GVL_Devices.VGP_80.Axis.PlcToNc <-> Inputs/FromPlc

CONFIGURATION plc_kfe_gatt
    RESOURCE PLC ON TwinCAT3
        TASK PlcTask(INTERVAL := T#10ms, PRIORITY := 20);
        PROGRAM PRG_1_PlcTask WITH PlcTask : PRG_1_PlcTask;
    END_RESOURCE
END_CONFIGURATION

// ---- DUTs/E_State.TcDUT
{attribute 'qualified_only'}
{attribute 'strict'}
TYPE E_State :
(
    unknown,
    error,
    warning,
    ok
);
END_TYPE

// ---- DUTs/E_GasType.TcDUT
TYPE E_GasType :
(
    none := 0,
    Nitrogen,
    Argon
);
END_TYPE

// ---- DUTs/E_HomeState.TcDUT
TYPE E_HomeState :
(
    H_READY,
    H_INIT,
    H_RESET_LL,
    H_RESET_HL,
    H_ENABLE,
    H_MOVING,
    H_MOVING2,
    H_CHECK,
    H_RESET,
    H_SET_POS,
    H_ERROR,
    H_WRITE_LL,
    H_WRITE_HL,
    H_DONE

) UDINT;
END_TYPE

// ---- DUTs/E_MAA_States.TcDUT
TYPE E_MAA_States :
(
    Unknown := 0,
    Aprt1 := 1, //smallest
    Aprt2 := 2,
    Aprt3 := 3,
    Aprt4 := 4,
	Centered:=5
);
END_TYPE

// ---- DUTs/E_MAA_States_X.TcDUT
TYPE E_MAA_States_X :
(
    Unknown := 0,
    Centered:=1
);
END_TYPE

// ---- DUTs/E_MoveState.TcDUT
TYPE E_MoveState :
(
    ABORT,
    INIT,
    ENABLE,
    FORWARD,
    BACKWARDS,
    READY,
    MOVING,
    NEWTARGETPOSITION,
    NEWTARGETPOSITION2,
    ERROR,
    RESET,
    HALT,
    HOME
) UDINT;
END_TYPE

// ---- DUTs/ST_DRL.TcDUT
TYPE ST_DRL :
STRUCT
    {attribute 'pytmc' := ' pv: TEMP '}
    TEMP AT%I*: UINT;
    {attribute 'pytmc' := ' pv: SV '}
    SV  AT%I*: UINT;
    {attribute 'pytmc' := ' pv: SC '}
    SC  AT%I*: UINT;
END_STRUCT
END_TYPE

// ---- DUTs/ST_VGP.TcDUT
TYPE ST_VGP :
STRUCT

    {attribute 'pytmc' := '
    pv: POS_RBV;
    io: i;
    '}
    // Inputs
    i_iPosition	:	REAL; //Encoder position readback (if it exists)
    {attribute 'pytmc' := '
    pv: ENC_RBV;
    io: i;
    '}
    // Inputs
    rEnoder_Position	:	REAL; //Encoder position readback (if it exists)
    {attribute 'pytmc' := '
    pv: ERROR;
    field: ZNAM FALSE;
     field: ONAM TRUE;
    io: i;
    '}
    // Inputs
    pv_xError	:	BOOL;

    {attribute 'pytmc' := '
    pv: IS_HOMED;
    field: ZNAM FALSE;
     field: ONAM TRUE;
    io: i;
    '}
    // Inputs
    pv_xHomed	:	BOOL :=false;


    //Softvariables
    {attribute 'pytmc' := '
    pv: ILK_OK;
    field: ZNAM FALSE;
     field: ONAM TRUE;
    io: i;
    '}
    xIlkOK	:	BOOL := FALSE; // Interlock Bit
    //Manually Pressing valve "Open/Close" on EDM
    {attribute 'pytmc' := '
    pv: OPN_SW;
    field: ZNAM FALSE;
     field: ONAM TRUE;
    io: io;
    '}
    pv_xOPN_SW	: BOOL;

    {attribute 'pytmc' := '
    pv: GO_SW;
    field: ZNAM FALSE;
    field: ONAM TRUE;
    io: io;
    '}
    pv_xGo_SW	: BOOL;

    {attribute 'pytmc' := '
    pv: HOME_SW;
    field: ZNAM FALSE;
     field: ONAM TRUE;
    io: io;
    '}
    pv_xHome_SW	: BOOL;

    {attribute 'pytmc' := '
    pv: Reset_SW;
    field: ZNAM FALSE;
     field: ONAM TRUE;
    io: io;
    '}
    pv_xReset_SW	: BOOL;

    {attribute 'pytmc' := '
    pv: Busy;
    field: ZNAM FALSE;
     field: ONAM TRUE;
    io: io;
    '}
    xBusy	: BOOL;

    {attribute 'pytmc' := '
    pv: ABORT;
     field: ZNAM FALSE;
     field: ONAM TRUE;
    io: io;
    '}
    pv_xABORT_SW	: BOOL;


    {attribute 'pytmc' := '
    pv: POS_CTRL;
    io: io;
    '}
    rReqPosition	:	REAL;
    // Outputs
    {attribute 'pytmc' := '
    pv: POS_DES;
    io: io;
    '}
    q_iRawPosition	:	INT; //Position control
    {attribute 'pytmc' := '
    pv: STATE;
    type: mbbi ;
    field: ZRST CLOSE ;
    field: ONST OPEN;
    field: TWST PRESS CNTRL ;
    field: THST MANUAL CNTRL ;
    io: io;
    '}
    eValveControl	:	E_VCN := CloseValve; // Valve control state
    /// state machine state
    {attribute 'pytmc' := '
    pv: Axis_STATE;
    io: io;
    '}
    eState: E_MoveState; //Axis Move state
    ftIlk	:	F_TRIG;
    {attribute 'pytmc' := '
    pv: ERR_ID;
    io: i;
    '}
    nErrorID: UDINT;

    {attribute 'pytmc' := '
    pv: ERR_MSG;
    io: i;
    '}
    sErrorMessage : STRING;

END_STRUCT
END_TYPE

// ---- Version/Global_Version.TcGVL
{attribute 'TcGenerated'}
{attribute 'no-analysis'}
{attribute 'linkalways'}
// This function has been automatically generated from the project information.
VAR_GLOBAL CONSTANT
    {attribute 'const_non_replaced'}
    stLibVersion_KFE_GATT : ST_LibVersion := (iMajor := 0, iMinor := 3, iBuild := 1, iRevision := 0, nFlags := 1, sVersion := '0.3.1');
END_VAR

// ---- GVLs/GVL_Devices.TcGVL
VAR_GLOBAL
(*AT1K0*)
/// Injector
//Valves
    {attribute 'pytmc' :=' pv: AT1K0:GAS:VCN:70 '}
    VCN_70 : FB_VCN;

    {attribute 'pytmc' :=' pv: AT1K0:GAS:VVC:71 '}
    VVC_71 : FB_VVC;

    {attribute 'pytmc' :=' pv: AT1K0:GAS:VVC:72 '}
    VVC_72 : FB_VVC;


    {attribute 'pytmc' :=' pv: AT1K0:GAS:VGP:80 '}
    VGP_80 : FB_VGP;

//Gauges
    {attribute 'pytmc' :=' pv: AT1K0:GAS:GCM:70 '}
    GCM_70: FB_GCM;
    {attribute 'pytmc' :=' pv: AT1K0:GAS:GCM:80 '}
    GCM_80: FB_GCM;
    {attribute 'pytmc' :=' pv: AT1K0:GAS:GCM:81 '}
    GCM_81: FB_GCM;
    (*Pseudo gauge device Structure to combine the readings of two GCM gauges*)
    {attribute 'pytmc' :=' pv: AT1K0:GAS:GCM:82  '}
    GCM_82 : ST_VG;


/////////////////////////////


    //////////////////////////////////
// MKS275 Gauges

{attribute 'pytmc' := ' pv: AT1K0:GAS:GPI:111 '}
fb_AT1K0_GAS_GPI_111 : FB_MKS275;
{attribute 'pytmc' := ' pv: AT1K0:GAS:GPI:121 '}
fb_AT1K0_GAS_GPI_121 : FB_MKS275;
{attribute 'pytmc' := ' pv: AT1K0:GAS:GPI:141 '}
fb_AT1K0_GAS_GPI_141 : FB_MKS275;

// FB_MKS317

{attribute 'pytmc' := ' pv: AT1K0:GAS:GPI:10 '}
fb_AT1K0_GAS_GPI_10 : FB_MKS317;
{attribute 'pytmc' := ' pv: AT1K0:GAS:GPI:20 '}
fb_AT1K0_GAS_GPI_20 : FB_MKS317;
{attribute 'pytmc' := ' pv: AT1K0:GAS:GPI:11 '}
fb_AT1K0_GAS_GPI_11 : FB_MKS317;
{attribute 'pytmc' := ' pv: AT1K0:GAS:GPI:30 '}
fb_AT1K0_GAS_GPI_30 : FB_MKS317;
{attribute 'pytmc' := ' pv: AT1K0:GAS:GPI:40 '}
fb_AT1K0_GAS_GPI_40 : FB_MKS317;
{attribute 'pytmc' := ' pv: AT1K0:GAS:GPI:50 '}
fb_AT1K0_GAS_GPI_50 : FB_MKS317;
{attribute 'pytmc' := ' pv: AT1K0:GAS:GPI:60 '}
fb_AT1K0_GAS_GPI_60 : FB_MKS317;
{attribute 'pytmc' := ' pv: AT1K0:GAS:GPI:51 '}
fb_AT1K0_GAS_GPI_51 : FB_MKS317;
{attribute 'pytmc' := ' pv: AT1K0:GAS:GPI:80 '}
fb_AT1K0_GAS_GPI_80 : FB_MKS317;
{attribute 'pytmc' := ' pv: AT1K0:GAS:GPI:90 '}
fb_AT1K0_GAS_GPI_90 : FB_MKS317;
{attribute 'pytmc' := ' pv: AT1K0:GAS:GPI:100 '}
fb_AT1K0_GAS_GPI_100 : FB_MKS317;
{attribute 'pytmc' := ' pv: AT1K0:GAS:GPI:110 '}
fb_AT1K0_GAS_GPI_110 : FB_MKS317;
{attribute 'pytmc' := ' pv: AT1K0:GAS:GPI:120 '}
fb_AT1K0_GAS_GPI_120 : FB_MKS317;
{attribute 'pytmc' := ' pv: AT1K0:GAS:GPI:130 '}
fb_AT1K0_GAS_GPI_130 : FB_MKS317;
{attribute 'pytmc' := ' pv: AT1K0:GAS:GPI:140 '}
fb_AT1K0_GAS_GPI_140 : FB_MKS317;

// FB_MKS422

{attribute 'pytmc' := ' pv: AT1K0:GAS:GCC:10 '}
fb_AT1K0_GAS_GCC_10 : FB_MKS422;
{attribute 'pytmc' := ' pv: AT1K0:GAS:GCC:20 '}
fb_AT1K0_GAS_GCC_20 : FB_MKS422;
{attribute 'pytmc' := ' pv: AT1K0:GAS:GCC:30 '}
fb_AT1K0_GAS_GCC_30 : FB_MKS422;
{attribute 'pytmc' := ' pv: AT1K0:GAS:GCC:40 '}
fb_AT1K0_GAS_GCC_40 : FB_MKS422;
{attribute 'pytmc' := ' pv: AT1K0:GAS:GCC:50 '}
fb_AT1K0_GAS_GCC_50 : FB_MKS422;
{attribute 'pytmc' := ' pv: AT1K0:GAS:GCC:60 '}
fb_AT1K0_GAS_GCC_60 : FB_MKS422;
{attribute 'pytmc' := ' pv: AT1K0:GAS:GCC:80 '}
fb_AT1K0_GAS_GCC_80 : FB_MKS422;
{attribute 'pytmc' := ' pv: AT1K0:GAS:GCC:90 '}
fb_AT1K0_GAS_GCC_90 : FB_MKS422;
{attribute 'pytmc' := ' pv: AT1K0:GAS:GCC:100 '}
fb_AT1K0_GAS_GCC_100 : FB_MKS422;
{attribute 'pytmc' := ' pv: AT1K0:GAS:GCC:110 '}
fb_AT1K0_GAS_GCC_110 : FB_MKS422;
{attribute 'pytmc' := ' pv: AT1K0:GAS:GCC:120 '}
fb_AT1K0_GAS_GCC_120 : FB_MKS422;
{attribute 'pytmc' := ' pv: AT1K0:GAS:GCC:130 '}
fb_AT1K0_GAS_GCC_130 : FB_MKS422;
{attribute 'pytmc' := ' pv: AT1K0:GAS:GCC:140 '}
fb_AT1K0_GAS_GCC_140 : FB_MKS422;




// FB_VRC

{attribute 'pytmc' := ' pv: AT1K0:GAS:VRC:10 '}
fb_AT1K0_GAS_VRC_10 : FB_VRC_EBD;
{attribute 'pytmc' := ' pv: AT1K0:GAS:VRC:20 '}
fb_AT1K0_GAS_VRC_20 : FB_VRC_EBD;
{attribute 'pytmc' := ' pv: AT1K0:GAS:VRC:30 '}
fb_AT1K0_GAS_VRC_30 : FB_VRC_EBD;
{attribute 'pytmc' := ' pv: AT1K0:GAS:VRC:40 '}
fb_AT1K0_GAS_VRC_40 : FB_VRC_EBD;
{attribute 'pytmc' := ' pv: AT1K0:GAS:VRC:50 '}
fb_AT1K0_GAS_VRC_50 : FB_VRC;
{attribute 'pytmc' := ' pv: AT1K0:GAS:VRC:60 '}
fb_AT1K0_GAS_VRC_60 : FB_VRC;
{attribute 'pytmc' := ' pv: AT1K0:GAS:VRC:70 '}
fb_AT1K0_GAS_VRC_70 : FB_VRC;
{attribute 'pytmc' := ' pv: AT1K0:GAS:VRC:80 '}
fb_AT1K0_GAS_VRC_80 : FB_VRC;
{attribute 'pytmc' := ' pv: AT1K0:GAS:VRC:90 '}
fb_AT1K0_GAS_VRC_90 : FB_VRC;
{attribute 'pytmc' := ' pv: AT1K0:GAS:VRC:100 '}
fb_AT1K0_GAS_VRC_100 : FB_VRC;
{attribute 'pytmc' := ' pv: AT1K0:GAS:VRC:110 '}
fb_AT1K0_GAS_VRC_110 : FB_VRC;
{attribute 'pytmc' := ' pv: AT1K0:GAS:VRC:120 '}
fb_AT1K0_GAS_VRC_120 : FB_VRC;
{attribute 'pytmc' := ' pv: AT1K0:GAS:VRC:130 '}
fb_AT1K0_GAS_VRC_130 : FB_VRC;
{attribute 'pytmc' := ' pv: AT1K0:GAS:VRC:140 '}
fb_AT1K0_GAS_VRC_140 : FB_VRC;

// PUMPS
// Turbos
// FB_PTM_Ebara_010M
{attribute 'pytmc' := ' pv: AT1K0:GAS:PTM:10 '}
fb_AT1K0_GAS_PTM_10 : FB_PTM_Ebara_010M;
{attribute 'pytmc' := ' pv: AT1K0:GAS:PTM:20 '}
fb_AT1K0_GAS_PTM_20 : FB_PTM_Ebara_010M;
{attribute 'pytmc' := ' pv: AT1K0:GAS:PTM:30 '}
fb_AT1K0_GAS_PTM_30 : FB_PTM_Ebara_010M;
{attribute 'pytmc' := ' pv: AT1K0:GAS:PTM:40 '}
fb_AT1K0_GAS_PTM_40 : FB_PTM_Ebara_010M;
{attribute 'pytmc' := ' pv: AT1K0:GAS:PTM:80 '}
fb_AT1K0_GAS_PTM_80 : FB_PTM_TwisTorr;
{attribute 'pytmc' := ' pv: AT1K0:GAS:PTM:120 '}
fb_AT1K0_GAS_PTM_120 : FB_PTM_Ebara_010M;
{attribute 'pytmc' := ' pv: AT1K0:GAS:PTM:130 '}
fb_AT1K0_GAS_PTM_130 : FB_PTM_Ebara_010M;
{attribute 'pytmc' := ' pv: AT1K0:GAS:PTM:140 '}
fb_AT1K0_GAS_PTM_140 : FB_PTM_Ebara_010M;
// FB_PTM_Ebara_011M
{attribute 'pytmc' := ' pv: AT1K0:GAS:PTM:110 '}
fb_AT1K0_GAS_PTM_110 : FB_PTM_Ebara_011M;

// Roughing
// FB_EbaraDryPump
{attribute 'pytmc' := ' pv: AT1K0:GAS:PMF:10 '}
fb_AT1K0_GAS_PMF_10 : FB_ScrollPump;
{attribute 'pytmc' := ' pv: AT1K0:GAS:PMF:60 '}
fb_AT1K0_GAS_PMF_60 : FB_ScrollPump;
{attribute 'pytmc' := ' pv: AT1K0:GAS:PMF:90 '}
fb_AT1K0_GAS_PMF_90 : FB_EbaraDryPump;
{attribute 'pytmc' := ' pv: AT1K0:GAS:PMF:100 '}
fb_AT1K0_GAS_PMF_100 : FB_EbaraDryPump;
{attribute 'pytmc' := ' pv: AT1K0:GAS:PMF:110 '}
fb_AT1K0_GAS_PMF_110 : FB_EbaraEVA;
{attribute 'pytmc' := ' pv: AT1K0:GAS:PMF:120 '}
fb_AT1K0_GAS_PMF_120 : FB_EbaraEVA;
{attribute 'pytmc' := ' pv: AT1K0:GAS:PMF:140 '}
fb_AT1K0_GAS_PMF_140 : FB_EbaraEVA;

//Roughing DC Valves
{attribute 'pytmc' := ' pv: AT1K0:GAS:VCP:110 '}
//{attribute 'TcLinkTo' := 	'.q_xOPN_DO	:=	TIIB[=+-EL2212_06_25]^DOX Control Channel 1^Control^Output'}
{attribute 'TcLinkTo' := 	'.q_xOPN_DO	:=	TIIB[=+-ES2004_05_02]^Channel 3^Output'}
fb_AT1K0_GAS_VVC_110 : FB_VVC;
{attribute 'pytmc' := ' pv: AT1K0:GAS:VCP:120 '}
//{attribute 'TcLinkTo' := 	'.q_xOPN_DO	:=	TIIB[=+-EL2212_06_25]^DOX Control Channel 2^Control^Output'}
{attribute 'TcLinkTo' := 	'.q_xOPN_DO	:=	TIIB[=+-ES2004_05_02]^Channel 4^Output'}
fb_AT1K0_GAS_VVC_120 : FB_VVC;
{attribute 'pytmc' := ' pv: AT1K0:GAS:VCP:140 '}
//{attribute 'TcLinkTo' := 	'.q_xOPN_DO	:=	TIIB[=+-EL2212_04_18]^DOX Control Channel 1^Control^Output'}
{attribute 'TcLinkTo' := 	'.q_xOPN_DO	:=	TIIB[=+-ES2004_05_04]^Channel 3^Output'}
fb_AT1K0_GAS_VVC_140 : FB_VVC;

//PTM 80 VRC back stream valve
{attribute 'pytmc' := ' pv: AT1K0:GAS:VVC:80 '}
{attribute 'TcLinkTo' := 	'.q_xOPN_DO	:=	TIIB[=+-EL2212_04_18]^DOX Control Channel 2^Control^Output'}
fb_AT1K0_GAS_VVC_80 : FB_VVC;
//NEW added Valve instead of the manual valve at the roughing line in the EBD
{attribute 'pytmc' := ' pv: AT1K0:GAS:VRC:11 '}
{attribute 'TcLinkTo' := 	'.q_xOPN_DO	:=	TIIB[=+-ES2008_02_14]^Channel 1^Output;
                            .i_xClsLS	:=	TIIB[=+-ES1004_03_21]^Channel 2^Input;
                            .i_xOpnLS	:=	TIIB[=+-ES1004_03_21]^Channel 1^Input'}


fb_AT1K0_GAS_VRC_11 : FB_VRC_EBD;

{attribute 'pytmc' := ' pv: AT1K0:GAS:GPI:12 '}
{attribute 'TcLinkTo' := 	'.i_iPRESS_R	:=	TIIB[=+-ES3064_01_09]^AI Standard Channel 4^Value'}
fb_AT1K0_GAS_GPI_12 : FB_MKS317;

END_VAR

// ---- GVLs/GVL_GATT.TcGVL
VAR_GLOBAL

fbLogHandler: FB_LogHandler;
fbLogger : FB_LogMessage := (eSubsystem:=E_SubSystem.MPS,nMinTimeViolationAcceptable:=10,nLocalTripThreshold := T#500ms);
fbEcatDiagWrapper : FB_EcatDiagWrapper;

END_VAR

// ---- GVLs/GVL_PMPS.TcGVL
VAR_GLOBAL

//MPS
    {attribute 'pytmc' := '
    pv: PLC:KFE:GATT:FFO:01
    '}
    {attribute 'TcLinkTo' := '.q_xFastFaultOut:=TIIB[=+-ES2202_00_07]^Channel 1^Output'}
    g_FastFaultOutput1  :   FB_HardwareFFOutput :=(i_sNetID:='172.21.92.73.1.1');

    {attribute 'pytmc' := '
    pv: PLC:KFE:GATT:FFO:02
    '}
    {attribute 'TcLinkTo' := '.q_xFastFaultOut:=TIIB[=+-ES2202_00_07]^Channel 2^Output'}
    g_FastFaultOutput2  :   FB_HardwareFFOutput :=(i_sNetID:='172.21.92.73.1.1');

    {attribute 'pytmc' := '
     pv: PLC:KFE:GATT:FF_RESET;
     field: ZNAM FALSE;
     field: ONAM TRUE;
     io: io;
    '}
    xFastFaultReset :   BOOL;
    {attribute 'pytmc' := '
    pv: PLC:KFE:GATT:ARB:01
    '}
    fbArbiter1   :   FB_Arbiter(1);
    {attribute 'pytmc' := '
    pv: PLC:KFE:GATT:ARB:02
    '}
    fbArbiter2   :   FB_Arbiter(2);

    {attribute 'pytmc' := '
    pv: AT1K0:GAS:MODE ;
     field: ZNAM Local;
    field: ONAM PMPS;
     io: io;
    '}
    xPMPSMode	:BOOL;

    {attribute 'TcLinkTo' := ':=TIIB[PMPS_PRE]^IO Inputs^Requested Transmission'}
    Req_Trans AT%I*: ST_PMPS_Attenuator_IO;

     {attribute 'TcLinkTo' := ':=TIIB[PMPS_PRE]^IO Outputs^Current Transmission'}
    Cur_Trans AT%Q*: ST_PMPS_Attenuator_IO;
    {attribute 'pytmc' := '
    pv: AT1K0:GAS:PhotonEnergy
    '}

    rPhotonEnergy : REAL;

    stStatus: ST_AttenuatorStatus;
    {attribute 'TcLinkTo' := ':=TIIB[PMPS_PRE]^IO Outputs^bGattStatus'}
    bStatus  AT%Q*:Byte;


END_VAR

// ---- GVLs/GVL_MOT.TcGVL
VAR_GLOBAL


END_VAR

// ---- GVLs/GVL_Variables.TcGVL
VAR_GLOBAL

